C09131=1138.833,163.232,-60.014,-178.582,7.169,148.928
C09132=1138.829,163.481,-60.036,-178.579,7.171,148.927
C09133=1138.824,163.730,-60.058,-178.576,7.174,148.927
C09134=1138.820,163.979,-60.080,-178.574,7.176,148.927
C09135=1138.815,164.228,-60.102,-178.571,7.177,148.926
C09136=1138.810,164.478,-60.124,-178.568,7.180,148.926
C09137=1138.805,164.726,-60.146,-178.565,7.182,148.926
C09138=1138.801,164.975,-60.169,-178.562,7.185,148.925
C09139=1138.796,165.224,-60.191,-178.560,7.186,148.925
C09140=1138.792,165.473,-60.213,-178.557,7.188,148.925
C09141=1138.787,165.722,-60.234,-178.554,7.191,148.924
C09142=1138.782,165.971,-60.257,-178.551,7.193,148.924
C09143=1138.777,166.220,-60.279,-178.548,7.195,148.924
C09144=1138.773,166.469,-60.301,-178.545,7.197,148.923
C09145=1138.769,166.717,-60.323,-178.543,7.200,148.923
C09146=1138.764,166.967,-60.346,-178.540,7.201,148.923
C09147=1138.759,167.216,-60.367,-178.537,7.203,148.923
C09148=1138.754,167.465,-60.390,-178.534,7.206,148.922
C09149=1138.750,167.714,-60.412,-178.532,7.208,148.922
C09150=1138.745,167.963,-60.435,-178.528,7.210,148.922
C09151=1138.741,168.212,-60.457,-178.526,7.212,148.921
C09152=1138.736,168.461,-60.478,-178.523,7.215,148.921
C09153=1138.731,168.710,-60.501,-178.520,7.217,148.921
C09154=1138.726,168.958,-60.523,-178.518,7.219,148.921
C09155=1138.722,169.208,-60.545,-178.515,7.221,148.920
C09156=1138.718,169.457,-60.567,-178.512,7.223,148.920
C09157=1138.712,169.705,-60.590,-178.509,7.226,148.920
C09158=1138.708,169.955,-60.612,-178.506,7.228,148.919
C09159=1138.703,170.203,-60.634,-178.503,7.230,148.919
C09160=1138.698,170.452,-60.657,-178.500,7.232,148.919
C09161=1138.694,170.702,-60.680,-178.497,7.235,148.919
C09162=1138.689,170.951,-60.702,-178.495,7.236,148.918
C09163=1138.685,171.199,-60.725,-178.492,7.239,148.918
C09164=1138.680,171.448,-60.746,-178.489,7.241,148.918
C09165=1138.675,171.697,-60.770,-178.487,7.243,148.917
C09166=1138.671,171.946,-60.792,-178.484,7.246,148.917
C09167=1138.665,172.195,-60.814,-178.481,7.247,148.917
C09168=1138.661,172.444,-60.837,-178.478,7.250,148.916
C09169=1138.657,172.693,-60.859,-178.475,7.252,148.916
C09170=1138.652,172.942,-60.882,-178.472,7.254,148.916
C09171=1138.647,173.191,-60.904,-178.469,7.256,148.916
C09172=1138.643,173.440,-60.927,-178.467,7.259,148.915
C09173=1138.638,173.689,-60.949,-178.464,7.261,148.915
C09174=1138.633,173.938,-60.972,-178.461,7.263,148.915
C09175=1138.629,174.187,-60.994,-178.458,7.265,148.915
C09176=1138.624,174.435,-61.017,-178.455,7.268,148.914
C09177=1138.620,174.684,-61.040,-178.452,7.270,148.914
C09178=1138.615,174.934,-61.063,-178.450,7.273,148.914
C09179=1138.610,175.182,-61.085,-178.447,7.274,148.913
C09180=1138.605,175.431,-61.108,-178.444,7.277,148.913
C09181=1138.601,175.680,-61.130,-178.441,7.279,148.913
C09182=1138.596,175.929,-61.154,-178.438,7.281,148.912
C09183=1138.591,176.178,-61.176,-178.436,7.284,148.912
C09184=1138.587,176.427,-61.199,-178.433,7.286,148.912
C09185=1138.583,176.676,-61.222,-178.430,7.288,148.912
C09186=1138.578,176.925,-61.244,-178.427,7.291,148.912
C09187=1138.573,177.173,-61.267,-178.424,7.292,148.911
C09188=1138.569,177.422,-61.290,-178.422,7.295,148.911
C09189=1138.563,177.672,-61.313,-178.419,7.297,148.911
C09190=1138.560,177.921,-61.335,-178.416,7.300,148.910
C09191=1138.554,178.169,-61.358,-178.413,7.302,148.910
C09192=1138.550,178.418,-61.381,-178.410,7.304,148.910
C09193=1138.545,178.667,-61.404,-178.408,7.306,148.910
C09194=1138.541,178.916,-61.427,-178.404,7.309,148.909
C09195=1138.537,179.165,-61.450,-178.402,7.310,148.909
C09196=1138.531,179.413,-61.473,-178.399,7.313,148.909
C09197=1138.527,179.662,-61.496,-178.396,7.315,148.908
C09198=1138.522,179.912,-61.518,-178.393,7.318,148.908
C09199=1138.518,180.161,-61.542,-178.390,7.321,148.908
C09200=1138.514,180.410,-61.564,-178.388,7.323,148.908
C09201=1138.509,180.659,-61.588,-178.385,7.325,148.907
C09202=1138.504,180.907,-61.611,-178.382,7.327,148.907
C09203=1138.499,181.156,-61.634,-178.379,7.330,148.907
C09204=1138.495,181.405,-61.657,-178.376,7.331,148.907
C09205=1138.490,181.654,-61.680,-178.374,7.334,148.907
C09206=1138.485,181.903,-61.703,-178.371,7.336,148.906
C09207=1138.481,182.152,-61.726,-178.368,7.339,148.906
C09208=1138.477,182.401,-61.749,-178.365,7.341,148.906
C09209=1138.471,182.649,-61.772,-178.362,7.343,148.905
C09210=1138.467,182.898,-61.795,-178.359,7.346,148.905
C09211=1138.462,183.167,-61.821,-178.357,7.348,148.905
C09212=1138.458,183.438,-61.846,-178.354,7.351,148.905
C09213=1138.452,183.708,-61.871,-178.350,7.353,148.904
C09214=1138.447,183.977,-61.896,-178.347,7.356,148.904
C09215=1138.442,184.226,-61.919,-178.344,7.359,148.904
C09216=1138.438,184.475,-61.942,-178.342,7.360,148.904
C09217=1138.434,184.724,-61.966,-178.339,7.363,148.903
C09218=1138.429,184.972,-61.990,-178.336,7.365,148.903
C09219=1138.424,185.221,-62.013,-178.333,7.368,148.903
C09220=1138.419,185.470,-62.036,-178.331,7.370,148.903
C09221=1138.415,185.719,-62.059,-178.327,7.372,148.902
C09222=1138.411,185.968,-62.082,-178.325,7.375,148.902
C09223=1138.406,186.217,-62.105,-178.322,7.377,148.902
C09224=1138.401,186.466,-62.129,-178.319,7.380,148.902
C09225=1138.396,186.715,-62.152,-178.316,7.381,148.901
C09226=1138.392,186.963,-62.176,-178.314,7.384,148.901
C09227=1138.387,187.212,-62.200,-178.310,7.387,148.901
C09228=1138.383,187.461,-62.223,-178.308,7.389,148.901
C09229=1138.378,187.710,-62.246,-178.305,7.392,148.900
C09230=1138.374,187.959,-62.270,-178.302,7.394,148.900
C09231=1138.369,188.208,-62.294,-178.299,7.396,148.900
C09232=1138.364,188.457,-62.317,-178.296,7.399,148.900
C09233=1138.360,188.706,-62.340,-178.294,7.401,148.899
C09234=1138.355,188.954,-62.365,-178.291,7.404,148.899
C09235=1138.350,189.203,-62.388,-178.288,7.405,148.899
C09236=1138.346,189.452,-62.411,-178.285,7.408,148.899
C09237=1138.341,189.701,-62.435,-178.282,7.411,148.898
C09238=1138.337,189.950,-62.459,-178.280,7.413,148.898
C09239=1138.332,190.199,-62.482,-178.277,7.415,148.898
C09240=1138.328,190.447,-62.506,-178.274,7.418,148.898
C09241=1138.323,190.696,-62.529,-178.271,7.420,148.898
C09242=1138.318,190.945,-62.553,-178.268,7.423,148.897
C09243=1138.314,191.194,-62.577,-178.266,7.425,148.897
C09244=1138.309,191.443,-62.600,-178.263,7.428,148.897
C09245=1138.305,191.691,-62.624,-178.259,7.430,148.897
C09246=1138.300,191.940,-62.648,-178.257,7.432,148.896
C09247=1138.295,192.189,-62.671,-178.254,7.435,148.896
C09248=1138.291,192.437,-62.695,-178.252,7.437,148.896
C09249=1138.287,192.687,-62.719,-178.248,7.439,148.896
C09250=1138.282,192.936,-62.743,-178.246,7.442,148.896
C09251=1138.278,193.185,-62.766,-178.243,7.444,148.895
C09252=1138.273,193.433,-62.790,-178.240,7.447,148.895
C09253=1138.268,193.682,-62.814,-178.237,7.450,148.895
C09254=1138.263,193.931,-62.838,-178.235,7.452,148.895
C09255=1138.259,194.180,-62.862,-178.232,7.454,148.894
C09256=1138.254,194.428,-62.886,-178.228,7.457,148.894
C09257=1138.250,194.677,-62.910,-178.226,7.459,148.894
C09258=1138.246,194.926,-62.934,-178.223,7.462,148.894
C09259=1138.241,195.175,-62.958,-178.220,7.464,148.894
C09260=1138.236,195.424,-62.982,-178.218,7.467,148.893
C09261=1138.232,195.673,-63.006,-178.215,7.469,148.893
C09262=1138.227,195.921,-63.030,-178.212,7.472,148.893
C09263=1138.223,196.170,-63.053,-178.209,7.474,148.893
C09264=1138.217,196.419,-63.078,-178.206,7.477,148.892
C09265=1138.214,196.668,-63.102,-178.203,7.479,148.892
C09266=1138.209,196.917,-63.126,-178.201,7.481,148.892
C09267=1138.205,197.165,-63.150,-178.198,7.484,148.892
C09268=1138.199,197.414,-63.174,-178.195,7.487,148.892
C09269=1138.195,197.662,-63.198,-178.193,7.489,148.891
C09270=1138.191,197.912,-63.222,-178.189,7.491,148.891
C09271=1138.186,198.161,-63.246,-178.186,7.494,148.891
C09272=1138.181,198.409,-63.271,-178.184,7.496,148.891
C09273=1138.177,198.658,-63.295,-178.181,7.499,148.891
C09274=1138.172,198.907,-63.318,-178.178,7.502,148.890
C09275=1138.168,199.156,-63.343,-178.175,7.504,148.890
C09276=1138.163,199.405,-63.367,-178.173,7.506,148.890
C09277=1138.159,199.653,-63.392,-178.169,7.509,148.890
C09278=1138.155,199.901,-63.416,-178.167,7.511,148.889
C09279=1138.150,200.151,-63.441,-178.164,7.514,148.889
C09280=1138.145,200.400,-63.464,-178.161,7.516,148.889
C09281=1138.140,200.649,-63.489,-178.159,7.519,148.889
C09282=1138.136,200.897,-63.513,-178.156,7.521,148.889
C09283=1138.132,201.146,-63.537,-178.153,7.524,148.888
C09284=1138.127,201.395,-63.562,-178.150,7.527,148.888
C09285=1138.122,201.643,-63.586,-178.147,7.529,148.888
C09286=1138.118,201.892,-63.610,-178.144,7.532,148.888
C09287=1138.114,202.141,-63.635,-178.142,7.534,148.888
C09288=1138.109,202.390,-63.659,-178.139,7.536,148.887
C09289=1138.104,202.638,-63.684,-178.136,7.539,148.887
C09290=1138.100,202.887,-63.708,-178.133,7.542,148.887
C09291=1138.095,203.136,-63.733,-178.130,7.545,148.887
C09292=1138.091,203.384,-63.757,-178.128,7.547,148.887
C09293=1138.087,203.634,-63.781,-178.125,7.550,148.887
C09294=1138.082,203.882,-63.806,-178.122,7.552,148.886
C09295=1138.077,204.131,-63.830,-178.119,7.555,148.886
C09296=1138.073,204.380,-63.855,-178.116,7.557,148.886
C09297=1138.068,204.629,-63.879,-178.113,7.560,148.886
C09298=1138.063,204.877,-63.904,-178.111,7.563,148.886
C09299=1138.060,205.126,-63.929,-178.108,7.564,148.885
C09300=1138.055,205.375,-63.954,-178.105,7.567,148.885
C09301=1138.050,205.623,-63.978,-178.102,7.570,148.885
C09302=1138.046,205.872,-64.003,-178.099,7.573,148.885
C09303=1138.041,206.121,-64.028,-178.097,7.575,148.885
C09304=1138.036,206.369,-64.052,-178.094,7.578,148.885
C09305=1138.032,206.619,-64.077,-178.091,7.580,148.884
C09306=1138.028,206.867,-64.101,-178.088,7.583,148.884
C09307=1138.023,207.116,-64.126,-178.086,7.585,148.884
C09308=1138.018,207.365,-64.151,-178.083,7.588,148.884
C09309=1138.014,207.613,-64.175,-178.080,7.591,148.884
C09310=1138.009,207.862,-64.201,-178.077,7.593,148.883
C09311=1138.005,208.110,-64.225,-178.074,7.596,148.883
C09312=1138.000,208.360,-64.250,-178.071,7.598,148.883
C09313=1137.996,208.608,-64.275,-178.068,7.601,148.883
C09314=1137.991,208.856,-64.300,-178.066,7.604,148.883
C09315=1137.986,209.128,-64.327,-178.062,7.606,148.882
C09316=1137.981,209.398,-64.354,-178.059,7.609,148.882
C09317=1137.976,209.669,-64.381,-178.056,7.612,148.882
C09318=1137.972,209.940,-64.408,-178.053,7.615,148.882
C09319=1137.967,210.188,-64.433,-178.051,7.618,148.882
C09320=1137.962,210.437,-64.459,-178.047,7.620,148.882
C09321=1137.958,210.685,-64.483,-178.045,7.622,148.881
C09322=1137.954,210.934,-64.508,-178.042,7.625,148.881
C09323=1137.949,211.183,-64.533,-178.039,7.628,148.881
C09324=1137.945,211.432,-64.557,-178.036,7.631,148.881
C09325=1137.940,211.680,-64.583,-178.033,7.634,148.881
C09326=1137.935,211.930,-64.608,-178.031,7.636,148.881
C09327=1137.931,212.178,-64.633,-178.028,7.639,148.881
C09328=1137.926,212.427,-64.658,-178.025,7.641,148.880
C09329=1137.922,212.675,-64.683,-178.022,7.644,148.880
C09330=1137.917,212.924,-64.708,-178.019,7.647,148.880
C09331=1137.913,213.172,-64.733,-178.017,7.649,148.880
C09332=1137.908,213.421,-64.759,-178.014,7.652,148.880
C09333=1137.904,213.670,-64.783,-178.011,7.655,148.879
C09334=1137.900,213.919,-64.809,-178.008,7.657,148.879
C09335=1137.895,214.168,-64.834,-178.006,7.660,148.879
C09336=1137.890,214.416,-64.859,-178.003,7.662,148.879
C09337=1137.886,214.665,-64.885,-178.000,7.665,148.879
C09338=1137.881,214.914,-64.910,-177.997,7.668,148.879
C09339=1137.877,215.162,-64.936,-177.994,7.671,148.879
C09340=1137.872,215.411,-64.960,-177.991,7.673,148.878
C09341=1137.868,215.660,-64.985,-177.988,7.676,148.878
C09342=1137.864,215.908,-65.011,-177.986,7.678,148.878
C09343=1137.859,216.156,-65.037,-177.983,7.681,148.878
C09344=1137.855,216.406,-65.062,-177.981,7.684,148.878
C09345=1137.850,216.654,-65.087,-177.977,7.687,148.878
C09346=1137.846,216.903,-65.113,-177.974,7.690,148.878
C09347=1137.841,217.152,-65.138,-177.972,7.692,148.877
C09348=1137.836,217.400,-65.163,-177.969,7.695,148.877
C09349=1137.832,217.649,-65.189,-177.966,7.697,148.877
C09350=1137.827,217.897,-65.214,-177.963,7.700,148.877
C09351=1137.823,218.146,-65.240,-177.961,7.703,148.877
C09352=1137.818,218.396,-65.265,-177.958,7.706,148.877
C09353=1137.814,218.643,-65.290,-177.955,7.709,148.877
C09354=1137.810,218.892,-65.316,-177.952,7.711,148.876
C09355=1137.806,219.141,-65.341,-177.949,7.713,148.876
C09356=1137.801,219.389,-65.367,-177.947,7.716,148.876
C09357=1137.797,219.638,-65.393,-177.944,7.719,148.876
C09358=1137.792,219.887,-65.419,-177.941,7.722,148.876
C09359=1137.787,220.135,-65.444,-177.938,7.725,148.876
C09360=1137.783,220.384,-65.469,-177.935,7.728,148.875
C09361=1137.778,220.633,-65.495,-177.933,7.730,148.875
C09362=1137.774,220.882,-65.521,-177.930,7.733,148.875
C09363=1137.769,221.130,-65.546,-177.927,7.735,148.875
C09364=1137.765,221.379,-65.572,-177.924,7.738,148.875
C09365=1137.761,221.628,-65.598,-177.921,7.741,148.875
C09366=1137.756,221.876,-65.623,-177.918,7.744,148.875
C09367=1137.752,222.125,-65.649,-177.915,7.747,148.875
C09368=1137.748,222.373,-65.675,-177.913,7.749,148.874
C09369=1137.743,222.622,-65.700,-177.910,7.752,148.874
C09370=1137.738,222.871,-65.726,-177.908,7.755,148.874
C09371=1137.734,223.119,-65.753,-177.905,7.758,148.874
C09372=1137.730,223.368,-65.779,-177.901,7.760,148.874
C09373=1137.725,223.616,-65.804,-177.899,7.763,148.874
C09374=1137.721,223.865,-65.830,-177.896,7.766,148.874
C09375=1137.716,224.113,-65.855,-177.893,7.769,148.874
C09376=1137.711,224.363,-65.882,-177.891,7.771,148.873
C09377=1137.707,224.611,-65.908,-177.888,7.774,148.873
C09378=1137.702,224.859,-65.933,-177.885,7.777,148.873
C09379=1137.698,225.108,-65.959,-177.882,7.780,148.873
C09380=1137.694,225.356,-65.985,-177.879,7.782,148.873
C09381=1137.689,225.606,-66.011,-177.876,7.785,148.873
C09382=1137.685,225.854,-66.037,-177.874,7.788,148.873
C09383=1137.680,226.102,-66.063,-177.871,7.791,148.873
C09384=1137.676,226.351,-66.089,-177.868,7.794,148.872
C09385=1137.671,226.600,-66.115,-177.865,7.797,148.872
C09386=1137.667,226.849,-66.141,-177.863,7.799,148.872
C09387=1137.663,227.097,-66.167,-177.860,7.802,148.872
C09388=1137.658,227.345,-66.194,-177.857,7.804,148.872
C09389=1137.653,227.594,-66.219,-177.854,7.807,148.872
C09390=1137.649,227.843,-66.245,-177.851,7.810,148.872
C09391=1137.645,228.091,-66.272,-177.848,7.813,148.872
C09392=1137.640,228.340,-66.298,-177.846,7.816,148.872
C09393=1137.636,228.589,-66.324,-177.843,7.819,148.871
C09394=1137.632,228.837,-66.350,-177.840,7.822,148.871
C09395=1137.627,229.086,-66.377,-177.837,7.825,148.871
C09396=1137.623,229.334,-66.403,-177.834,7.828,148.871
C09397=1137.618,229.583,-66.429,-177.832,7.830,148.871
C09398=1137.613,229.832,-66.455,-177.829,7.833,148.871
C09399=1137.609,230.080,-66.481,-177.826,7.835,148.871
C09400=1137.605,230.329,-66.508,-177.823,7.838,148.871
C09401=1137.601,230.577,-66.534,-177.821,7.841,148.870
C09402=1137.596,230.826,-66.560,-177.818,7.844,148.870
C09403=1137.592,231.074,-66.587,-177.815,7.847,148.870
C09404=1137.587,231.323,-66.613,-177.812,7.850,148.870
C09405=1137.583,231.572,-66.640,-177.809,7.853,148.870
C09406=1137.579,231.820,-66.665,-177.806,7.855,148.870
C09407=1137.573,232.068,-66.692,-177.804,7.858,148.870
C09408=1137.569,232.316,-66.719,-177.801,7.861,148.870
C09409=1137.564,232.566,-66.745,-177.798,7.864,148.870
C09410=1137.561,232.814,-66.771,-177.795,7.867,148.870
C09411=1137.556,233.063,-66.798,-177.792,7.870,148.870
C09412=1137.552,233.311,-66.824,-177.790,7.873,148.870
C09413=1137.547,233.560,-66.851,-177.787,7.876,148.869
C09414=1137.543,233.808,-66.877,-177.784,7.879,148.869
C09415=1137.538,234.057,-66.904,-177.782,7.881,148.869
C09416=1137.534,234.305,-66.930,-177.779,7.883,148.869
C09417=1137.529,234.554,-66.957,-177.776,7.886,148.869
C09418=1137.525,234.802,-66.983,-177.773,7.889,148.869
C09419=1137.521,235.075,-67.013,-177.770,7.893,148.869
C09420=1137.515,235.347,-67.042,-177.767,7.896,148.869
C09421=1137.510,235.618,-67.071,-177.764,7.899,148.869
C09422=1137.506,235.890,-67.100,-177.761,7.902,148.869
C09423=1137.502,236.139,-67.127,-177.758,7.905,148.868
C09424=1137.497,236.388,-67.154,-177.755,7.908,148.868
C09425=1137.493,236.636,-67.180,-177.752,7.911,148.868
C09426=1137.488,236.885,-67.207,-177.749,7.914,148.868
C09427=1137.484,237.133,-67.234,-177.747,7.917,148.868
C09428=1137.480,237.381,-67.261,-177.744,7.920,148.868
C09429=1137.475,237.630,-67.288,-177.741,7.923,148.868
C09430=1137.470,237.879,-67.314,-177.738,7.926,148.868
C09431=1137.466,238.127,-67.340,-177.736,7.928,148.868
C09432=1137.461,238.376,-67.368,-177.733,7.931,148.868
C09433=1137.457,238.624,-67.395,-177.730,7.934,148.868
C09434=1137.453,238.872,-67.421,-177.728,7.937,148.867
C09435=1137.448,239.121,-67.448,-177.725,7.940,148.867
C09436=1137.444,239.369,-67.475,-177.722,7.942,148.867
C09437=1137.440,239.618,-67.502,-177.719,7.945,148.867
C09438=1137.436,239.867,-67.529,-177.716,7.948,148.867
C09439=1137.431,240.115,-67.556,-177.714,7.951,148.867
C09440=1137.426,240.364,-67.583,-177.711,7.954,148.867
C09441=1137.422,240.612,-67.610,-177.708,7.957,148.867
C09442=1137.418,240.860,-67.637,-177.705,7.960,148.867
C09443=1137.413,241.109,-67.664,-177.702,7.963,148.867
C09444=1137.409,241.358,-67.691,-177.700,7.966,148.867
C09445=1137.404,241.607,-67.718,-177.697,7.969,148.867
C09446=1137.400,241.855,-67.745,-177.694,7.972,148.867
C09447=1137.396,242.103,-67.772,-177.691,7.974,148.866
C09448=1137.391,242.352,-67.799,-177.688,7.977,148.866
C09449=1137.387,242.600,-67.827,-177.686,7.980,148.866
C09450=1137.383,242.849,-67.854,-177.682,7.984,148.866
C09451=1137.378,243.097,-67.881,-177.679,7.987,148.866
C09452=1137.374,243.346,-67.908,-177.677,7.990,148.866
C09453=1137.370,243.594,-67.935,-177.674,7.993,148.866
C09454=1137.365,243.843,-67.962,-177.671,7.996,148.866
C09455=1137.361,244.091,-67.990,-177.668,7.999,148.866
C09456=1137.356,244.340,-68.017,-177.666,8.002,148.866
C09457=1137.352,244.588,-68.044,-177.663,8.005,148.866
C09458=1137.347,244.837,-68.071,-177.660,8.008,148.866
C09459=1137.343,245.084,-68.099,-177.657,8.011,148.866
C09460=1137.339,245.334,-68.126,-177.655,8.013,148.866
C09461=1137.334,245.582,-68.153,-177.652,8.016,148.866
C09462=1137.329,245.831,-68.180,-177.649,8.019,148.866
C09463=1137.325,246.079,-68.208,-177.646,8.022,148.865
C09464=1137.322,246.327,-68.235,-177.643,8.025,148.865
C09465=1137.317,246.576,-68.262,-177.641,8.028,148.865
C09466=1137.313,246.824,-68.290,-177.638,8.031,148.865
C09467=1137.308,247.072,-68.317,-177.635,8.034,148.865
C09468=1137.304,247.321,-68.345,-177.632,8.037,148.865
C09469=1137.300,247.569,-68.372,-177.629,8.040,148.865
C09470=1137.294,247.818,-68.400,-177.627,8.043,148.865
C09471=1137.291,248.067,-68.428,-177.624,8.046,148.865
C09472=1137.286,248.315,-68.455,-177.621,8.049,148.865
C09473=1137.282,248.563,-68.483,-177.619,8.052,148.865
C09474=1137.277,248.812,-68.510,-177.616,8.055,148.865
C09475=1137.273,249.060,-68.538,-177.613,8.057,148.865
C09476=1137.268,249.309,-68.565,-177.610,8.061,148.865
C09477=1137.264,249.557,-68.593,-177.607,8.064,148.865
C09478=1137.260,249.806,-68.620,-177.604,8.067,148.865
C09479=1137.256,250.054,-68.648,-177.601,8.070,148.864
C09480=1137.252,250.303,-68.675,-177.599,8.073,148.865
C09481=1137.247,250.551,-68.703,-177.596,8.076,148.865
C09482=1137.243,250.799,-68.730,-177.593,8.079,148.864
C09483=1137.238,251.048,-68.759,-177.590,8.082,148.864
C09484=1137.234,251.296,-68.787,-177.588,8.085,148.864
C09485=1137.229,251.544,-68.814,-177.585,8.088,148.864
C09486=1137.225,251.793,-68.842,-177.582,8.091,148.864
C09487=1137.221,252.041,-68.870,-177.579,8.094,148.864
C09488=1137.216,252.289,-68.897,-177.577,8.097,148.864
C09489=1137.212,252.538,-68.926,-177.574,8.100,148.864
C09490=1137.208,252.786,-68.953,-177.571,8.103,148.864
C09491=1137.203,253.035,-68.981,-177.568,8.106,148.864
C09492=1137.199,253.283,-69.009,-177.565,8.109,148.864
C09493=1137.195,253.532,-69.037,-177.562,8.112,148.864
C09494=1137.190,253.781,-69.064,-177.560,8.115,148.864
C09495=1137.186,254.028,-69.092,-177.557,8.118,148.864
C09496=1137.182,254.277,-69.120,-177.554,8.121,148.864
C09497=1137.178,254.525,-69.148,-177.552,8.124,148.864
C09498=1137.173,254.774,-69.177,-177.549,8.127,148.864
C09499=1137.168,255.022,-69.204,-177.546,8.130,148.864
C09500=1137.165,255.271,-69.232,-177.543,8.133,148.864
C09501=1137.160,255.519,-69.260,-177.540,8.137,148.864
C09502=1137.156,255.768,-69.288,-177.538,8.140,148.864
C09503=1137.151,256.016,-69.316,-177.535,8.143,148.864
C09504=1137.146,256.264,-69.345,-177.532,8.146,148.864
C09505=1137.143,256.512,-69.373,-177.529,8.149,148.864
C09506=1137.138,256.760,-69.401,-177.526,8.152,148.864
C09507=1137.133,257.010,-69.429,-177.524,8.155,148.864
C09508=1137.129,257.258,-69.456,-177.521,8.158,148.864
C09509=1137.125,257.506,-69.484,-177.518,8.161,148.864
C09510=1137.120,257.754,-69.513,-177.515,8.164,148.863
C09511=1137.117,258.003,-69.541,-177.512,8.167,148.863
C09512=1137.112,258.252,-69.570,-177.510,8.171,148.864
C09513=1137.108,258.500,-69.597,-177.507,8.174,148.863
C09514=1137.104,258.748,-69.626,-177.504,8.176,148.863
C09515=1137.099,258.996,-69.654,-177.501,8.179,148.863
C09516=1137.095,259.245,-69.682,-177.499,8.182,148.863
C09517=1137.090,259.493,-69.711,-177.496,8.186,148.863
C09518=1137.087,259.741,-69.739,-177.493,8.189,148.863
C09519=1137.081,259.989,-69.768,-177.490,8.192,148.863
C09520=1137.078,260.238,-69.796,-177.487,8.195,148.863
C09521=1137.073,260.486,-69.824,-177.485,8.198,148.863
C09522=1137.069,260.735,-69.852,-177.482,8.201,148.863
C09523=1137.064,261.008,-69.883,-177.479,8.205,148.863
C09524=1137.060,261.282,-69.915,-177.476,8.208,148.863
C09525=1137.054,261.555,-69.947,-177.473,8.212,148.863
C09526=1137.050,261.829,-69.978,-177.470,8.215,148.863
C09527=1137.045,262.078,-70.006,-177.467,8.218,148.863
C09528=1137.042,262.326,-70.035,-177.464,8.222,148.863
C09529=1137.037,262.574,-70.063,-177.461,8.224,148.863
C09530=1137.033,262.822,-70.092,-177.459,8.227,148.863
C09531=1137.028,263.071,-70.120,-177.456,8.231,148.863
C09532=1137.024,263.318,-70.149,-177.453,8.234,148.863
C09533=1137.020,263.567,-70.177,-177.451,8.236,148.863
C09534=1137.015,263.816,-70.206,-177.447,8.240,148.863
C09535=1137.011,264.063,-70.235,-177.445,8.243,148.863
C09536=1137.007,264.312,-70.263,-177.442,8.246,148.863
C09537=1137.002,264.561,-70.292,-177.439,8.249,148.863
C09538=1136.998,264.809,-70.321,-177.436,8.252,148.863
C09539=1136.994,265.057,-70.349,-177.434,8.255,148.863
C09540=1136.990,265.306,-70.378,-177.431,8.258,148.863
C09541=1136.985,265.554,-70.407,-177.428,8.262,148.863
C09542=1136.981,265.802,-70.435,-177.425,8.265,148.863
C09543=1136.977,266.051,-70.465,-177.423,8.268,148.863
C09544=1136.972,266.299,-70.493,-177.420,8.271,148.863
C09545=1136.968,266.547,-70.522,-177.417,8.274,148.863
C09546=1136.964,266.796,-70.551,-177.414,8.278,148.863
C09547=1136.959,267.044,-70.579,-177.411,8.281,148.863
C09548=1136.955,267.292,-70.608,-177.409,8.284,148.863
C09549=1136.951,267.541,-70.637,-177.406,8.287,148.863
C09550=1136.946,267.789,-70.666,-177.404,8.290,148.863
C09551=1136.942,268.036,-70.695,-177.401,8.293,148.863
C09552=1136.938,268.285,-70.723,-177.397,8.297,148.863
C09553=1136.934,268.533,-70.753,-177.395,8.300,148.863
C09554=1136.929,268.782,-70.782,-177.392,8.303,148.863
C09555=1136.925,269.030,-70.810,-177.389,8.306,148.863
C09556=1136.921,269.278,-70.840,-177.387,8.309,148.863
C09557=1136.917,269.527,-70.868,-177.384,8.313,148.863
C09558=1136.912,269.775,-70.898,-177.381,8.316,148.863
C09559=1136.907,270.023,-70.926,-177.379,8.319,148.863
C09560=1136.903,270.271,-70.956,-177.376,8.322,148.863
C09561=1136.900,270.519,-70.984,-177.373,8.325,148.863
C09562=1136.895,270.768,-71.014,-177.370,8.329,148.864
C09563=1136.891,271.017,-71.043,-177.367,8.332,148.863
C09564=1136.886,271.264,-71.072,-177.364,8.335,148.863
C09565=1136.882,271.512,-71.101,-177.362,8.338,148.864
C09566=1136.877,271.761,-71.130,-177.359,8.341,148.864
C09567=1136.873,272.010,-71.159,-177.356,8.345,148.863
C09568=1136.869,272.258,-71.189,-177.354,8.348,148.864
C09569=1136.866,272.506,-71.218,-177.351,8.351,148.864
C09570=1136.861,272.753,-71.247,-177.348,8.354,148.864
C09571=1136.857,273.002,-71.276,-177.346,8.357,148.864
C09572=1136.852,273.251,-71.305,-177.342,8.361,148.864
C09573=1136.848,273.499,-71.334,-177.339,8.364,148.864
C09574=1136.844,273.747,-71.364,-177.337,8.367,148.864
C09575=1136.840,273.995,-71.393,-177.334,8.370,148.864
C09576=1136.836,274.244,-71.423,-177.331,8.374,148.864
C09577=1136.831,274.492,-71.452,-177.329,8.377,148.864
C09578=1136.827,274.739,-71.481,-177.326,8.380,148.864
C09579=1136.822,274.988,-71.511,-177.323,8.383,148.864
C09580=1136.818,275.236,-71.540,-177.320,8.387,148.864
C09581=1136.814,275.484,-71.570,-177.317,8.390,148.864
C09582=1136.810,275.732,-71.599,-177.315,8.393,148.864
C09583=1136.806,275.981,-71.629,-177.312,8.396,148.864
C09584=1136.801,276.229,-71.658,-177.310,8.399,148.864
C09585=1136.797,276.477,-71.688,-177.306,8.403,148.864
C09586=1136.793,276.726,-71.717,-177.304,8.406,148.864
C09587=1136.789,276.974,-71.746,-177.301,8.409,148.864
C09588=1136.784,277.222,-71.776,-177.299,8.412,148.864
C09589=1136.780,277.471,-71.806,-177.296,8.416,148.864
C09590=1136.776,277.719,-71.835,-177.293,8.419,148.864
C09591=1136.771,277.967,-71.865,-177.290,8.422,148.864
C09592=1136.767,278.215,-71.894,-177.288,8.425,148.864
C09593=1136.763,278.464,-71.924,-177.284,8.429,148.864
C09594=1136.759,278.711,-71.954,-177.282,8.432,148.865
C09595=1136.755,278.960,-71.983,-177.279,8.435,148.865
C09596=1136.751,279.208,-72.013,-177.277,8.438,148.865
C09597=1136.746,279.457,-72.043,-177.273,8.442,148.865
C09598=1136.742,279.705,-72.072,-177.271,8.445,148.865
C09599=1136.738,279.952,-72.102,-177.268,8.448,148.865
C09600=1136.734,280.201,-72.132,-177.265,8.452,148.865
C09601=1136.730,280.449,-72.161,-177.263,8.455,148.865
C09602=1136.725,280.698,-72.191,-177.260,8.458,148.865
C09603=1136.721,280.945,-72.222,-177.257,8.461,148.865
C09604=1136.717,281.193,-72.251,-177.254,8.465,148.865
C09605=1136.712,281.442,-72.281,-177.252,8.468,148.865
C09606=1136.708,281.690,-72.311,-177.249,8.471,148.865
C09607=1136.704,281.938,-72.341,-177.247,8.475,148.865
C09608=1136.699,282.186,-72.370,-177.243,8.478,148.865
C09609=1136.695,282.434,-72.400,-177.241,8.481,148.865
C09610=1136.691,282.682,-72.430,-177.238,8.484,148.865
C09611=1136.686,282.931,-72.460,-177.235,8.488,148.866
C09612=1136.683,283.178,-72.490,-177.232,8.491,148.866
C09613=1136.678,283.427,-72.520,-177.230,8.495,148.866
C09614=1136.674,283.675,-72.550,-177.227,8.498,148.866
C09615=1136.670,283.923,-72.580,-177.224,8.502,148.866
C09616=1136.666,284.172,-72.611,-177.221,8.505,148.866
C09617=1136.661,284.420,-72.640,-177.219,8.508,148.866
C09618=1136.657,284.667,-72.670,-177.216,8.512,148.866
C09619=1136.653,284.916,-72.700,-177.213,8.515,148.866
C09620=1136.649,285.164,-72.731,-177.211,8.518,148.866
C09621=1136.644,285.412,-72.761,-177.208,8.522,148.866
C09622=1136.640,285.660,-72.791,-177.205,8.525,148.866
C09623=1136.636,285.908,-72.820,-177.203,8.528,148.866
C09624=1136.632,286.157,-72.851,-177.200,8.531,148.866
C09625=1136.628,286.404,-72.882,-177.197,8.535,148.867
C09626=1136.623,286.653,-72.912,-177.194,8.538,148.866
C09627=1136.619,286.928,-72.945,-177.191,8.542,148.867
C09628=1136.613,287.204,-72.979,-177.188,8.546,148.867
C09629=1136.609,287.480,-73.012,-177.185,8.549,148.867
C09630=1136.604,287.755,-73.047,-177.182,8.553,148.867
C09631=1136.600,288.004,-73.076,-177.179,8.557,148.867
C09632=1136.596,288.252,-73.107,-177.176,8.560,148.867
C09633=1136.592,288.499,-73.137,-177.174,8.563,148.867
C09634=1136.588,288.748,-73.168,-177.171,8.567,148.867
C09635=1136.583,288.996,-73.197,-177.168,8.570,148.867
C09636=1136.579,289.244,-73.228,-177.166,8.573,148.867
C09637=1136.575,289.492,-73.258,-177.162,8.577,148.867
C09638=1136.570,289.740,-73.289,-177.160,8.580,148.868
C09639=1136.567,289.988,-73.320,-177.157,8.583,148.868
C09640=1136.562,290.237,-73.350,-177.154,8.587,148.868
C09641=1136.558,290.484,-73.380,-177.152,8.590,148.868
C09642=1136.554,290.732,-73.411,-177.149,8.593,148.868
C09643=1136.550,290.981,-73.442,-177.146,8.597,148.868
C09644=1136.546,291.229,-73.472,-177.144,8.600,148.868
C09645=1136.541,291.477,-73.503,-177.141,8.604,148.868
C09646=1136.538,291.725,-73.533,-177.138,8.608,148.868
C09647=1136.533,291.973,-73.564,-177.135,8.611,148.868
C09648=1136.529,292.221,-73.595,-177.133,8.614,148.869
C09649=1136.525,292.469,-73.624,-177.130,8.618,148.869
C09650=1136.521,292.718,-73.655,-177.127,8.621,148.869
C09651=1136.516,292.966,-73.686,-177.125,8.624,148.869
C09652=1136.512,293.213,-73.716,-177.122,8.628,148.869
C09653=1136.508,293.462,-73.747,-177.119,8.631,148.869
C09654=1136.503,293.710,-73.778,-177.117,8.634,148.869
C09655=1136.500,293.957,-73.809,-177.114,8.638,148.869
C09656=1136.496,294.206,-73.840,-177.111,8.641,148.869
C09657=1136.491,294.454,-73.871,-177.108,8.645,148.870
C09658=1136.487,294.701,-73.901,-177.106,8.648,148.870
C09659=1136.483,294.950,-73.932,-177.103,8.652,148.870
C09660=1136.479,295.198,-73.963,-177.100,8.656,148.870
C09661=1136.474,295.446,-73.994,-177.097,8.659,148.870
C09662=1136.471,295.694,-74.024,-177.095,8.662,148.870
C09663=1136.466,295.942,-74.055,-177.092,8.666,148.870
C09664=1136.462,296.190,-74.087,-177.089,8.669,148.870
C09665=1136.458,296.438,-74.118,-177.086,8.673,148.870
C09666=1136.453,296.686,-74.149,-177.084,8.676,148.871
C09667=1136.450,296.935,-74.179,-177.081,8.679,148.871
C09668=1136.445,297.182,-74.210,-177.078,8.683,148.871
C09669=1136.442,297.430,-74.242,-177.076,8.686,148.871
C09670=1136.437,297.678,-74.272,-177.073,8.689,148.871
C09671=1136.432,297.926,-74.303,-177.070,8.693,148.871
C09672=1136.428,298.175,-74.334,-177.068,8.697,148.871
C09673=1136.424,298.422,-74.366,-177.065,8.700,148.871
C09674=1136.421,298.671,-74.396,-177.062,8.704,148.871
C09675=1136.416,298.919,-74.427,-177.060,8.707,148.872
C09676=1136.413,299.167,-74.459,-177.057,8.711,148.872
C09677=1136.408,299.415,-74.490,-177.054,8.714,148.872
C09678=1136.403,299.663,-74.520,-177.051,8.718,148.872
C09679=1136.400,299.911,-74.552,-177.049,8.721,148.872
C09680=1136.395,300.159,-74.583,-177.047,8.724,148.872
C09681=1136.391,300.407,-74.615,-177.043,8.728,148.872
C09682=1136.387,300.655,-74.646,-177.041,8.731,148.873
C09683=1136.383,300.903,-74.678,-177.038,8.735,148.873
C09684=1136.378,301.151,-74.708,-177.036,8.739,148.873
C09685=1136.374,301.399,-74.739,-177.032,8.742,148.873
C09686=1136.370,301.647,-74.771,-177.030,8.746,148.873
C09687=1136.366,301.895,-74.802,-177.028,8.749,148.873
C09688=1136.362,302.143,-74.834,-177.025,8.753,148.873
C09689=1136.358,302.391,-74.865,-177.022,8.756,148.873
C09690=1136.353,302.639,-74.896,-177.019,8.760,148.874
C09691=1136.350,302.887,-74.928,-177.017,8.763,148.874
C09692=1136.345,303.135,-74.959,-177.014,8.767,148.874
C09693=1136.341,303.383,-74.991,-177.011,8.770,148.874
C09694=1136.337,303.631,-75.021,-177.008,8.774,148.874
C09695=1136.333,303.879,-75.053,-177.006,8.778,148.874
C09696=1136.329,304.126,-75.085,-177.003,8.781,148.875
C09697=1136.325,304.375,-75.116,-177.000,8.785,148.875
C09698=1136.321,304.623,-75.148,-176.997,8.788,148.875
C09699=1136.316,304.870,-75.180,-176.995,8.792,148.875
C09700=1136.312,305.119,-75.211,-176.992,8.795,148.875
C09701=1136.308,305.366,-75.242,-176.990,8.798,148.875
C09702=1136.304,305.614,-75.274,-176.987,8.803,148.876
C09703=1136.286,306.680,-75.412,-177.856,10.498,149.535
C09704=1136.282,306.928,-75.444,-177.853,10.501,149.535
C09705=1136.278,307.176,-75.477,-177.850,10.503,149.535
C09706=1136.273,307.423,-75.508,-177.847,10.506,149.534
C09707=1136.270,307.671,-75.541,-177.844,10.509,149.534
C09708=1136.266,307.923,-75.574,-177.841,10.511,149.534
C09709=1136.261,308.174,-75.606,-177.837,10.513,149.534
C09710=1136.257,308.426,-75.639,-177.834,10.516,149.534
C09711=1136.253,308.678,-75.671,-177.831,10.519,149.533
C09712=1136.249,308.925,-75.703,-177.828,10.521,149.533
C09713=1136.245,309.173,-75.736,-177.825,10.524,149.533
C09714=1136.241,309.421,-75.767,-177.821,10.526,149.533
C09715=1136.236,309.669,-75.800,-177.819,10.529,149.533
C09716=1136.232,309.917,-75.832,-177.815,10.531,149.532
C09717=1136.228,310.165,-75.865,-177.812,10.534,149.532
C09718=1136.225,310.413,-75.897,-177.809,10.537,149.532
C09719=1136.220,310.660,-75.929,-177.806,10.539,149.532
C09720=1136.216,310.908,-75.961,-177.803,10.542,149.532
C09721=1136.212,311.156,-75.994,-177.799,10.544,149.531
C09722=1136.208,311.404,-76.026,-177.796,10.547,149.531
C09723=1136.204,311.652,-76.059,-177.793,10.550,149.531
C09724=1136.200,311.900,-76.091,-177.790,10.552,149.531
C09725=1136.195,312.148,-76.123,-177.787,10.555,149.531
C09726=1136.192,312.395,-76.155,-177.783,10.557,149.530
C09727=1136.187,312.643,-76.188,-177.781,10.560,149.530
C09728=1136.184,312.891,-76.220,-177.778,10.562,149.530
C09729=1136.179,313.139,-76.253,-177.775,10.564,149.530
C09730=1136.176,313.387,-76.285,-177.772,10.567,149.530
C09731=1136.172,313.635,-76.318,-177.768,10.569,149.530
C09732=1136.167,313.883,-76.350,-177.765,10.572,149.529
C09733=1136.163,314.130,-76.382,-177.762,10.574,149.529
C09734=1136.159,314.378,-76.415,-177.759,10.577,149.529
C09735=1136.155,314.626,-76.447,-177.756,10.580,149.529
C09736=1136.151,314.874,-76.480,-177.752,10.582,149.529
C09737=1136.147,315.122,-76.513,-177.749,10.585,149.529
C09738=1136.143,315.369,-76.545,-177.746,10.587,149.528
C09739=1136.139,315.618,-76.578,-177.743,10.590,149.528
C09740=1136.135,315.865,-76.611,-177.740,10.593,149.528
C09741=1136.131,316.113,-76.643,-177.737,10.595,149.528
C09742=1136.127,316.361,-76.676,-177.733,10.597,149.527
C09743=1136.123,316.609,-76.709,-177.730,10.600,149.527
C09744=1136.119,316.857,-76.741,-177.727,10.603,149.527
C09745=1136.115,317.105,-76.774,-177.724,10.605,149.527
C09746=1136.110,317.352,-76.807,-177.721,10.608,149.527
C09747=1136.106,317.600,-76.839,-177.717,10.610,149.527
C09748=1136.102,317.847,-76.872,-177.714,10.613,149.526
C09749=1136.098,318.095,-76.905,-177.711,10.615,149.526
C09750=1136.094,318.344,-76.938,-177.708,10.618,149.526
C09751=1136.090,318.591,-76.971,-177.705,10.621,149.526
C09752=1136.086,318.839,-77.003,-177.702,10.622,149.526
C09753=1136.082,319.086,-77.036,-177.699,10.625,149.525
C09754=1136.078,319.334,-77.070,-177.696,10.628,149.525
C09755=1136.073,319.582,-77.102,-177.693,10.630,149.525
C09756=1136.069,319.830,-77.135,-177.689,10.632,149.525
C09757=1136.066,320.078,-77.168,-177.686,10.635,149.525
C09758=1136.062,320.325,-77.201,-177.683,10.638,149.524
C09759=1136.058,320.574,-77.234,-177.680,10.640,149.524
C09760=1136.054,320.787,-77.263,-177.677,10.643,149.524
C09761=1136.051,321.001,-77.291,-177.674,10.645,149.524
C09762=1136.048,321.214,-77.320,-177.672,10.647,149.524
C09763=1136.044,321.428,-77.348,-177.669,10.649,149.524
C09764=1136.040,321.641,-77.376,-177.666,10.651,149.523
C09765=1136.038,321.855,-77.405,-177.663,10.654,149.523
C09766=1136.034,322.068,-77.433,-177.661,10.655,149.523
C09767=1136.030,322.282,-77.461,-177.658,10.658,149.523
C09768=1136.026,322.529,-77.495,-177.654,10.661,149.523
C09769=1136.022,322.777,-77.528,-177.651,10.663,149.523
C09770=1136.018,323.026,-77.561,-177.649,10.665,149.522
C09771=1136.014,323.273,-77.594,-177.645,10.667,149.522
C09772=1136.010,323.521,-77.628,-177.642,10.670,149.522
C09773=1136.006,323.769,-77.661,-177.639,10.673,149.522
C09774=1136.002,324.016,-77.695,-177.636,10.675,149.522
C09775=1135.998,324.264,-77.728,-177.633,10.678,149.522
C09776=1135.994,324.511,-77.761,-177.630,10.680,149.521
C09777=1135.990,324.759,-77.794,-177.626,10.683,149.521
C09778=1135.986,325.007,-77.827,-177.623,10.685,149.521
C09779=1135.982,325.255,-77.861,-177.620,10.688,149.521
C09780=1135.978,325.503,-77.894,-177.617,10.690,149.520
C09781=1135.974,325.751,-77.927,-177.613,10.693,149.520
C09782=1135.970,325.998,-77.961,-177.610,10.696,149.520
C09783=1135.966,326.246,-77.994,-177.607,10.698,149.520
C09784=1135.962,326.493,-78.027,-177.604,10.701,149.520
C09785=1135.958,326.742,-78.061,-177.601,10.703,149.520
C09786=1135.954,326.989,-78.094,-177.598,10.706,149.519
C09787=1135.950,327.237,-78.128,-177.594,10.708,149.519
C09788=1135.946,327.484,-78.161,-177.591,10.711,149.519
C09789=1135.942,327.732,-78.194,-177.588,10.713,149.519
C09790=1135.938,327.979,-78.228,-177.585,10.716,149.519
C09791=1135.934,328.228,-78.262,-177.581,10.718,149.518
C09792=1135.930,328.476,-78.295,-177.578,10.721,149.518
C09793=1135.925,328.723,-78.328,-177.575,10.724,149.518
C09794=1135.922,328.970,-78.362,-177.572,10.726,149.518
C09795=1135.918,329.218,-78.395,-177.568,10.728,149.518
C09796=1135.914,329.466,-78.430,-177.565,10.731,149.517
C09797=1135.910,329.714,-78.463,-177.562,10.734,149.517
C09798=1135.905,329.962,-78.497,-177.559,10.736,149.517
C09799=1135.901,330.209,-78.530,-177.556,10.739,149.517
C09800=1135.898,330.457,-78.564,-177.553,10.741,149.517
C09801=1135.894,330.704,-78.598,-177.549,10.744,149.516
C09802=1135.890,330.952,-78.631,-177.546,10.746,149.516
C09803=1135.885,331.200,-78.665,-177.543,10.749,149.516
C09804=1135.882,331.448,-78.699,-177.540,10.751,149.516
C09805=1135.878,331.695,-78.733,-177.537,10.753,149.516
C09806=1135.874,331.943,-78.766,-177.534,10.756,149.515
C09807=1135.869,332.190,-78.800,-177.530,10.758,149.515
C09808=1135.866,332.439,-78.834,-177.527,10.761,149.515
C09809=1135.862,332.686,-78.868,-177.524,10.763,149.515
C09810=1135.858,332.933,-78.901,-177.521,10.766,149.515
C09811=1135.854,333.182,-78.936,-177.517,10.768,149.514
C09812=1135.850,333.429,-78.970,-177.515,10.771,149.514
C09813=1135.846,333.676,-79.003,-177.511,10.773,149.514
C09814=1135.842,333.925,-79.038,-177.508,10.776,149.514
C09815=1135.838,334.172,-79.072,-177.505,10.778,149.514
C09816=1135.835,334.385,-79.100,-177.502,10.781,149.513
C09817=1135.831,334.598,-79.130,-177.499,10.783,149.513
C09818=1135.828,334.812,-79.160,-177.496,10.786,149.513
C09819=1135.824,335.025,-79.188,-177.493,10.787,149.513
C09820=1135.821,335.239,-79.218,-177.491,10.789,149.513
C09821=1135.817,335.452,-79.247,-177.488,10.792,149.513
C09822=1135.814,335.665,-79.276,-177.485,10.794,149.512
C09823=1135.810,335.879,-79.306,-177.482,10.796,149.512
C09824=1135.807,336.126,-79.340,-177.479,10.799,149.512
C09825=1135.803,336.374,-79.373,-177.476,10.801,149.512
C09826=1135.799,336.622,-79.408,-177.473,10.804,149.512
C09827=1135.795,336.869,-79.442,-177.469,10.806,149.511
C09828=1135.790,337.117,-79.476,-177.466,10.809,149.511
C09829=1135.787,337.365,-79.511,-177.463,10.811,149.511
C09830=1135.782,337.613,-79.544,-177.460,10.814,149.511
C09831=1135.779,337.860,-79.579,-177.456,10.816,149.511
C09832=1135.774,338.108,-79.613,-177.453,10.819,149.510
C09833=1135.771,338.355,-79.647,-177.450,10.821,149.510
C09834=1135.767,338.603,-79.682,-177.447,10.823,149.510
C09835=1135.763,338.850,-79.716,-177.444,10.826,149.510
C09836=1135.759,339.098,-79.751,-177.441,10.828,149.510
C09837=1135.755,339.345,-79.784,-177.438,10.831,149.509
C09838=1135.751,339.593,-79.819,-177.434,10.833,149.509
C09839=1135.747,339.841,-79.853,-177.431,10.836,149.509
C09840=1135.743,340.088,-79.888,-177.428,10.838,149.509
C09841=1135.739,340.336,-79.922,-177.425,10.841,149.509
C09842=1135.735,340.583,-79.956,-177.421,10.843,149.508
C09843=1135.731,340.831,-79.991,-177.418,10.846,149.508
C09844=1135.727,341.078,-80.025,-177.415,10.848,149.508
C09845=1135.723,341.327,-80.060,-177.411,10.851,149.508
C09846=1135.719,341.574,-80.094,-177.408,10.853,149.507
C09847=1135.715,341.822,-80.129,-177.405,10.856,149.507
C09848=1135.711,342.069,-80.163,-177.402,10.858,149.507
C09849=1135.707,342.317,-80.197,-177.399,10.861,149.507
C09850=1135.703,342.564,-80.232,-177.395,10.863,149.507
C09851=1135.699,342.812,-80.267,-177.392,10.866,149.506
C09852=1135.695,343.059,-80.301,-177.389,10.868,149.506
C09853=1135.691,343.307,-80.336,-177.386,10.871,149.506
C09854=1135.687,343.555,-80.370,-177.382,10.873,149.506
C09855=1135.684,343.802,-80.405,-177.379,10.876,149.506
C09856=1135.679,344.049,-80.440,-177.376,10.878,149.506
C09857=1135.675,344.297,-80.475,-177.372,10.881,149.505
C09858=1135.672,344.544,-80.509,-177.369,10.883,149.505
C09859=1135.668,344.792,-80.544,-177.366,10.886,149.505
C09860=1135.664,345.040,-80.579,-177.363,10.888,149.505
C09861=1135.659,345.287,-80.613,-177.360,10.891,149.505
C09862=1135.656,345.535,-80.648,-177.356,10.893,149.504
C09863=1135.652,345.782,-80.683,-177.353,10.896,149.504
C09864=1135.648,346.030,-80.718,-177.350,10.898,149.504
C09865=1135.644,346.277,-80.753,-177.346,10.901,149.504
C09866=1135.640,346.525,-80.787,-177.343,10.903,149.503
C09867=1135.636,346.773,-80.822,-177.340,10.906,149.503
C09868=1135.632,347.020,-80.857,-177.337,10.908,149.503
C09869=1135.628,347.268,-80.892,-177.333,10.911,149.503
C09870=1135.624,347.515,-80.927,-177.330,10.913,149.503
C09871=1135.621,347.762,-80.961,-177.327,10.916,149.502
C09872=1135.617,347.976,-80.992,-177.324,10.917,149.502
C09873=1135.614,348.190,-81.022,-177.321,10.920,149.502
C09874=1135.610,348.402,-81.052,-177.319,10.922,149.502
C09875=1135.607,348.615,-81.082,-177.315,10.924,149.502
C09876=1135.604,348.828,-81.112,-177.313,10.926,149.502
C09877=1135.600,349.042,-81.142,-177.310,10.929,149.501
C09878=1135.597,349.256,-81.173,-177.307,10.931,149.501
C09879=1135.593,349.468,-81.203,-177.305,10.933,149.501
C09880=1135.590,349.716,-81.237,-177.301,10.936,149.501
C09881=1135.586,349.964,-81.273,-177.297,10.938,149.500
C09882=1135.582,350.210,-81.308,-177.293,10.941,149.500
C09883=1135.578,350.458,-81.343,-177.289,10.944,149.500
C09884=1135.574,350.706,-81.378,-177.285,10.947,149.500
C09885=1135.570,350.954,-81.413,-177.281,10.950,149.499
C09886=1135.566,351.201,-81.448,-177.278,10.952,149.499
C09887=1135.562,351.448,-81.484,-177.274,10.954,149.499
C09888=1135.558,351.696,-81.519,-177.270,10.958,149.499
C09889=1135.554,351.943,-81.554,-177.267,10.960,149.498
C09890=1135.550,352.191,-81.590,-177.263,10.963,149.498
C09891=1135.547,352.438,-81.625,-177.260,10.965,149.498
C09892=1135.543,352.686,-81.661,-177.256,10.969,149.498
C09893=1135.538,352.933,-81.695,-177.252,10.971,149.497
C09894=1135.535,353.181,-81.731,-177.249,10.973,149.497
C09895=1135.531,353.428,-81.766,-177.245,10.977,149.497
C09896=1135.527,353.676,-81.802,-177.241,10.979,149.496
C09897=1135.523,353.923,-81.837,-177.238,10.981,149.496
C09898=1135.519,354.170,-81.872,-177.234,10.984,149.496
C09899=1135.515,354.418,-81.907,-177.230,10.986,149.495
C09900=1135.512,354.666,-81.943,-177.227,10.989,149.495
C09901=1135.508,354.913,-81.978,-177.223,10.992,149.495
C09902=1135.503,355.160,-82.014,-177.219,10.994,149.495
C09903=1135.499,355.408,-82.050,-177.216,10.997,149.494
C09904=1135.496,355.655,-82.085,-177.212,11.000,149.494
C09905=1135.492,355.903,-82.121,-177.208,11.002,149.494
C09906=1135.488,356.150,-82.156,-177.205,11.005,149.494
C09907=1135.485,356.398,-82.192,-177.201,11.007,149.493
C09908=1135.481,356.645,-82.227,-177.197,11.010,149.493
C09909=1135.477,356.892,-82.263,-177.194,11.012,149.493
C09910=1135.472,357.140,-82.299,-177.190,11.015,149.493
C09911=1135.469,357.387,-82.334,-177.187,11.017,149.492
C09912=1135.465,357.635,-82.370,-177.183,11.020,149.492
C09913=1135.462,357.882,-82.406,-177.180,11.022,149.492
C09914=1135.458,358.129,-82.442,-177.176,11.025,149.491
C09915=1135.453,358.376,-82.477,-177.173,11.027,149.491
C09916=1135.449,358.624,-82.513,-177.169,11.030,149.491
C09917=1135.446,358.871,-82.549,-177.166,11.032,149.491
C09918=1135.442,359.119,-82.584,-177.162,11.034,149.490
C09919=1135.438,359.366,-82.621,-177.159,11.037,149.490
C09920=1135.434,359.614,-82.656,-177.156,11.039,149.490
C09921=1135.431,359.861,-82.692,-177.152,11.042,149.490
C09922=1135.427,360.109,-82.728,-177.149,11.044,149.489
C09923=1135.423,360.356,-82.764,-177.145,11.046,149.489
C09924=1135.419,360.603,-82.800,-177.141,11.050,149.489
C09925=1135.416,360.851,-82.836,-177.138,11.052,149.488
C09926=1135.411,361.099,-82.872,-177.134,11.054,149.488
C09927=1135.408,361.345,-82.908,-177.131,11.057,149.488
C09928=1135.405,361.559,-82.939,-177.128,11.058,149.488
C09929=1135.401,361.771,-82.970,-177.125,11.061,149.488
C09930=1135.398,361.985,-83.000,-177.122,11.063,149.487
C09931=1135.394,362.198,-83.032,-177.120,11.064,149.487
C09932=1135.391,362.411,-83.063,-177.116,11.067,149.487
C09933=1135.388,362.624,-83.094,-177.114,11.069,149.487
C09934=1135.385,362.837,-83.125,-177.111,11.071,149.487
C09935=1135.382,363.050,-83.156,-177.108,11.073,149.486
C09936=1135.377,363.297,-83.192,-177.105,11.075,149.486
C09937=1135.374,363.544,-83.228,-177.101,11.078,149.486
C09938=1135.369,363.792,-83.264,-177.098,11.080,149.485
C09939=1135.366,364.040,-83.300,-177.095,11.083,149.485
C09940=1135.362,364.286,-83.336,-177.091,11.085,149.485
C09941=1135.358,364.534,-83.372,-177.089,11.087,149.485
C09942=1135.355,364.781,-83.409,-177.085,11.089,149.485
C09943=1135.350,365.028,-83.446,-177.082,11.092,149.484
C09944=1135.347,365.276,-83.481,-177.078,11.094,149.484
C09945=1135.343,365.523,-83.518,-177.075,11.096,149.484
C09946=1135.339,365.770,-83.553,-177.072,11.099,149.483
C09947=1135.335,366.018,-83.590,-177.068,11.101,149.483
C09948=1135.331,366.265,-83.626,-177.066,11.103,149.483
C09949=1135.328,366.513,-83.663,-177.062,11.105,149.483
C09950=1135.324,366.760,-83.699,-177.059,11.108,149.483
C09951=1135.320,367.008,-83.736,-177.056,11.110,149.482
C09952=1135.317,367.255,-83.772,-177.052,11.113,149.482
C09953=1135.313,367.502,-83.809,-177.050,11.114,149.482
C09954=1135.308,367.750,-83.845,-177.046,11.117,149.482
C09955=1135.305,367.997,-83.881,-177.043,11.119,149.482
C09956=1135.301,368.244,-83.918,-177.040,11.122,149.481
C09957=1135.297,368.491,-83.954,-177.037,11.124,149.481
C09958=1135.293,368.738,-83.990,-177.034,11.126,149.481
C09959=1135.289,368.986,-84.027,-177.031,11.129,149.481
C09960=1135.286,369.233,-84.064,-177.027,11.131,149.480
C09961=1135.282,369.480,-84.101,-177.025,11.133,149.480
C09962=1135.279,369.727,-84.137,-177.021,11.135,149.480
C09963=1135.274,369.975,-84.173,-177.018,11.138,149.480
C09964=1135.270,370.222,-84.210,-177.015,11.139,149.479
C09965=1135.267,370.469,-84.246,-177.012,11.142,149.479
C09966=1135.263,370.716,-84.283,-177.009,11.144,149.479
C09967=1135.259,370.963,-84.320,-177.006,11.146,149.479
C09968=1135.256,371.211,-84.357,-177.003,11.149,149.479
C09969=1135.252,371.458,-84.393,-177.000,11.151,149.479
C09970=1135.247,371.706,-84.430,-176.997,11.153,149.478
C09971=1135.244,371.953,-84.466,-176.994,11.155,149.478
C09972=1135.240,372.200,-84.503,-176.991,11.158,149.478
C09973=1135.236,372.448,-84.540,-176.988,11.160,149.478
C09974=1135.232,372.695,-84.577,-176.985,11.162,149.478
C09975=1135.229,372.942,-84.613,-176.982,11.164,149.477
C09976=1135.225,373.189,-84.650,-176.979,11.167,149.477
C09977=1135.221,373.436,-84.687,-176.977,11.169,149.477
C09978=1135.217,373.684,-84.724,-176.973,11.171,149.477
C09979=1135.214,373.931,-84.760,-176.970,11.174,149.477
C09980=1135.210,374.178,-84.797,-176.968,11.176,149.477
C09981=1135.206,374.426,-84.834,-176.965,11.178,149.476
C09982=1135.202,374.672,-84.871,-176.962,11.180,149.476
C09983=1135.199,374.920,-84.908,-176.959,11.183,149.476
C09984=1135.195,375.133,-84.940,-176.956,11.184,149.476
C09985=1135.192,375.346,-84.972,-176.954,11.186,149.476
C09986=1135.189,375.558,-85.003,-176.952,11.188,149.476
C09987=1135.185,375.772,-85.035,-176.949,11.190,149.476
C09988=1135.182,375.985,-85.067,-176.947,11.192,149.476
C09989=1135.179,376.197,-85.099,-176.945,11.194,149.475
C09990=1135.176,376.410,-85.131,-176.942,11.196,149.475
C09991=1135.173,376.623,-85.163,-176.940,11.198,149.475
C09992=1135.169,376.871,-85.200,-176.937,11.199,149.475
C09993=1135.165,377.118,-85.236,-176.934,11.202,149.475
C09994=1135.161,377.365,-85.274,-176.931,11.204,149.475
C09995=1135.158,377.612,-85.311,-176.928,11.207,149.475
C09996=1135.154,377.859,-85.348,-176.926,11.209,149.475
//INST
///DATE 2021/06/25 14:31
///ATTR SC,RW,RJ
////FRAME ROBOT
///GROUP1 RB1
NOP
MOVL C00000 V=800.0 PL=0
MOVL C00001 V=800.0 PL=0
MOVL C00002 V=800.0 PL=0
MOVL C00003 V=800.0 PL=0
MOVL C00004 V=800.0 PL=0
MOVL C00005 V=800.0 PL=0
MOVL C00006 V=800.0 PL=0
MOVL C00007 V=800.0 PL=0
MOVL C00008 V=800.0 PL=0
MOVL C00009 V=800.0 PL=0
MOVL C00010 V=800.0 PL=0
MOVL C00011 V=800.0 PL=0
MOVL C00012 V=800.0 PL=0
MOVL C00013 V=800.0 PL=0
MOVL C00014 V=800.0 PL=0
MOVL C00015 V=800.0 PL=0
MOVL C00016 V=800.0 PL=0
MOVL C00017 V=800.0 PL=0
MOVL C00018 V=800.0 PL=0
MOVL C00019 V=800.0 PL=0
MOVL C00020 V=800.0 PL=0
MOVL C00021 V=800.0 PL=0
MOVL C00022 V=800.0 PL=0
MOVL C00023 V=800.0 PL=0
MOVL C00024 V=800.0 PL=0
MOVL C00025 V=800.0 PL=0
MOVL C00026 V=800.0 PL=0
MOVL C00027 V=800.0 PL=0
MOVL C00028 V=800.0 PL=0
MOVL C00029 V=800.0 PL=0
MOVL C00030 V=800.0 PL=0
MOVL C00031 V=800.0 PL=0
MOVL C00032 V=800.0 PL=0
MOVL C00033 V=800.0 PL=0
MOVL C00034 V=800.0 PL=0
MOVL C00035 V=800.0 PL=0
MOVL C00036 V=800.0 PL=0
MOVL C00037 V=800.0 PL=0
MOVL C00038 V=800.0 PL=0
MOVL C00039 V=800.0 PL=0
MOVL C00040 V=800.0 PL=0
MOVL C00041 V=800.0 PL=0
MOVL C00042 V=800.0 PL=0
MOVL C00043 V=800.0 PL=0
MOVL C00044 V=800.0 PL=0
MOVL C00045 V=800.0 PL=0
MOVL C00046 V=800.0 PL=0
MOVL C00047 V=800.0 PL=0
MOVL C00048 V=800.0 PL=0
MOVL C00049 V=800.0 PL=0
MOVL C00050 V=800.0 PL=0
MOVL C00051 V=800.0 PL=0
MOVL C00052 V=800.0 PL=0
MOVL C00053 V=800.0 PL=0
MOVL C00054 V=800.0 PL=0
MOVL C00055 V=800.0 PL=0
MOVL C00056 V=800.0 PL=0
MOVL C00057 V=800.0 PL=0
MOVL C00058 V=800.0 PL=0
MOVL C00059 V=800.0 PL=0
MOVL C00060 V=800.0 PL=0
MOVL C00061 V=800.0 PL=0
MOVL C00062 V=800.0 PL=0
MOVL C00063 V=800.0 PL=0
MOVL C00064 V=800.0 PL=0
MOVL C00065 V=800.0 PL=0
MOVL C00066 V=800.0 PL=0
MOVL C00067 V=800.0 PL=0
MOVL C00068 V=800.0 PL=0
MOVL C00069 V=800.0 PL=0
MOVL C00070 V=800.0 PL=0
MOVL C00071 V=800.0 PL=0
MOVL C00072 V=800.0 PL=0
MOVL C00073 V=800.0 PL=0
MOVL C00074 V=800.0 PL=0
MOVL C00075 V=800.0 PL=0
MOVL C00076 V=800.0 PL=0
MOVL C00077 V=800.0 PL=0
MOVL C00078 V=800.0 PL=0
MOVL C00079 V=800.0 PL=0
MOVL C00080 V=800.0 PL=0
MOVL C00081 V=800.0 PL=0
MOVL C00082 V=800.0 PL=0
MOVL C00083 V=800.0 PL=0
MOVL C00084 V=800.0 PL=0
MOVL C00085 V=800.0 PL=0
MOVL C00086 V=800.0 PL=0
MOVL C00087 V=800.0 PL=0
MOVL C00088 V=800.0 PL=0
MOVL C00089 V=800.0 PL=0
MOVL C00090 V=800.0 PL=0
MOVL C00091 V=800.0 PL=0
MOVL C00092 V=800.0 PL=0
MOVL C00093 V=800.0 PL=0
MOVL C00094 V=800.0 PL=0
MOVL C00095 V=800.0 PL=0
MOVL C00096 V=800.0 PL=0
MOVL C00097 V=800.0 PL=0
MOVL C00098 V=800.0 PL=0
MOVL C00099 V=800.0 PL=0
MOVL C00100 V=800.0 PL=0
MOVL C00101 V=800.0 PL=0
MOVL C00102 V=800.0 PL=0
MOVL C00103 V=800.0 PL=0
MOVL C00104 V=800.0 PL=0
MOVL C00105 V=800.0 PL=0
MOVL C00106 V=800.0 PL=0
MOVL C00107 V=800.0 PL=0
MOVL C00108 V=800.0 PL=0
MOVL C00109 V=800.0 PL=0
MOVL C00110 V=800.0 PL=0
MOVL C00111 V=800.0 PL=0
MOVL C00112 V=800.0 PL=0
MOVL C00113 V=800.0 PL=0
MOVL C00114 V=800.0 PL=0
MOVL C00115 V=800.0 PL=0
MOVL C00116 V=800.0 PL=0
MOVL C00117 V=800.0 PL=0
MOVL C00118 V=800.0 PL=0
MOVL C00119 V=800.0 PL=0
MOVL C00120 V=800.0 PL=0
MOVL C00121 V=800.0 PL=0
MOVL C00122 V=800.0 PL=0
MOVL C00123 V=800.0 PL=0
MOVL C00124 V=800.0 PL=0
MOVL C00125 V=800.0 PL=0
MOVL C00126 V=800.0 PL=0
MOVL C00127 V=800.0 PL=0
MOVL C00128 V=800.0 PL=0
MOVL C00129 V=800.0 PL=0
MOVL C00130 V=800.0 PL=0
MOVL C00131 V=800.0 PL=0
MOVL C00132 V=800.0 PL=0
MOVL C00133 V=800.0 PL=0
MOVL C00134 V=800.0 PL=0
MOVL C00135 V=800.0 PL=0
MOVL C00136 V=800.0 PL=0
MOVL C00137 V=800.0 PL=0
MOVL C00138 V=800.0 PL=0
MOVL C00139 V=800.0 PL=0
MOVL C00140 V=800.0 PL=0
MOVL C00141 V=800.0 PL=0
MOVL C00142 V=800.0 PL=0
MOVL C00143 V=800.0 PL=0
MOVL C00144 V=800.0 PL=0
MOVL C00145 V=800.0 PL=0
MOVL C00146 V=800.0 PL=0
MOVL C00147 V=800.0 PL=0
MOVL C00148 V=800.0 PL=0
MOVL C00149 V=800.0 PL=0
MOVL C00150 V=800.0 PL=0
MOVL C00151 V=800.0 PL=0
MOVL C00152 V=800.0 PL=0
MOVL C00153 V=800.0 PL=0
MOVL C00154 V=800.0 PL=0
MOVL C00155 V=800.0 PL=0
MOVL C00156 V=800.0 PL=0
MOVL C00157 V=800.0 PL=0
MOVL C00158 V=800.0 PL=0
MOVL C00159 V=800.0 PL=0
MOVL C00160 V=800.0 PL=0
MOVL C00161 V=800.0 PL=0
MOVL C00162 V=800.0 PL=0
MOVL C00163 V=800.0 PL=0
MOVL C00164 V=800.0 PL=0
MOVL C00165 V=800.0 PL=0
MOVL C00166 V=800.0 PL=0
MOVL C00167 V=800.0 PL=0
MOVL C00168 V=800.0 PL=0
MOVL C00169 V=800.0 PL=0
MOVL C00170 V=800.0 PL=0
MOVL C00171 V=800.0 PL=0
MOVL C00172 V=800.0 PL=0
MOVL C00173 V=800.0 PL=0
MOVL C00174 V=800.0 PL=0
MOVL C00175 V=800.0 PL=0
MOVL C00176 V=800.0 PL=0
MOVL C00177 V=800.0 PL=0
MOVL C00178 V=800.0 PL=0
MOVL C00179 V=800.0 PL=0
MOVL C00180 V=800.0 PL=0
MOVL C00181 V=800.0 PL=0
MOVL C00182 V=800.0 PL=0
MOVL C00183 V=800.0 PL=0
MOVL C00184 V=800.0 PL=0
MOVL C00185 V=800.0 PL=0
MOVL C00186 V=800.0 PL=0
MOVL C00187 V=800.0 PL=0
MOVL C00188 V=800.0 PL=0
MOVL C00189 V=800.0 PL=0
MOVL C00190 V=800.0 PL=0
MOVL C00191 V=800.0 PL=0
MOVL C00192 V=800.0 PL=0
MOVL C00193 V=800.0 PL=0
MOVL C00194 V=800.0 PL=0
MOVL C00195 V=800.0 PL=0
MOVL C00196 V=800.0 PL=0
MOVL C00197 V=800.0 PL=0
MOVL C00198 V=800.0 PL=0
MOVL C00199 V=800.0 PL=0
MOVL C00200 V=800.0 PL=0
MOVL C00201 V=800.0 PL=0
MOVL C00202 V=800.0 PL=0
MOVL C00203 V=800.0 PL=0
MOVL C00204 V=800.0 PL=0
MOVL C00205 V=800.0 PL=0
MOVL C00206 V=800.0 PL=0
MOVL C00207 V=800.0 PL=0
MOVL C00208 V=800.0 PL=0
MOVL C00209 V=800.0 PL=0
MOVL C00210 V=800.0 PL=0
MOVL C00211 V=800.0 PL=0
MOVL C00212 V=800.0 PL=0
MOVL C00213 V=800.0 PL=0
MOVL C00214 V=800.0 PL=0
MOVL C00215 V=800.0 PL=0
MOVL C00216 V=800.0 PL=0
MOVL C00217 V=800.0 PL=0
MOVL C00218 V=800.0 PL=0
MOVL C00219 V=800.0 PL=0
MOVL C00220 V=800.0 PL=0
MOVL C00221 V=800.0 PL=0
MOVL C00222 V=800.0 PL=0
MOVL C00223 V=800.0 PL=0
MOVL C00224 V=800.0 PL=0
MOVL C00225 V=800.0 PL=0
MOVL C00226 V=800.0 PL=0
MOVL C00227 V=800.0 PL=0
MOVL C00228 V=800.0 PL=0
MOVL C00229 V=800.0 PL=0
MOVL C00230 V=800.0 PL=0
MOVL C00231 V=800.0 PL=0
MOVL C00232 V=800.0 PL=0
MOVL C00233 V=800.0 PL=0
MOVL C00234 V=800.0 PL=0
MOVL C00235 V=800.0 PL=0
MOVL C00236 V=800.0 PL=0
MOVL C00237 V=800.0 PL=0
MOVL C00238 V=800.0 PL=0
MOVL C00239 V=800.0 PL=0
MOVL C00240 V=800.0 PL=0
MOVL C00241 V=800.0 PL=0
MOVL C00242 V=800.0 PL=0
MOVL C00243 V=800.0 PL=0
MOVL C00244 V=800.0 PL=0
MOVL C00245 V=800.0 PL=0
MOVL C00246 V=800.0 PL=0
MOVL C00247 V=800.0 PL=0
MOVL C00248 V=800.0 PL=0
MOVL C00249 V=800.0 PL=0
MOVL C00250 V=800.0 PL=0
MOVL C00251 V=800.0 PL=0
MOVL C00252 V=800.0 PL=0
MOVL C00253 V=800.0 PL=0
MOVL C00254 V=800.0 PL=0
MOVL C00255 V=800.0 PL=0
MOVL C00256 V=800.0 PL=0
MOVL C00257 V=800.0 PL=0
MOVL C00258 V=800.0 PL=0
MOVL C00259 V=800.0 PL=0
MOVL C00260 V=800.0 PL=0
MOVL C00261 V=800.0 PL=0
MOVL C00262 V=800.0 PL=0
MOVL C00263 V=800.0 PL=0
MOVL C00264 V=800.0 PL=0
MOVL C00265 V=800.0 PL=0
MOVL C00266 V=800.0 PL=0
MOVL C00267 V=800.0 PL=0
MOVL C00268 V=800.0 PL=0
MOVL C00269 V=800.0 PL=0
MOVL C00270 V=800.0 PL=0
MOVL C00271 V=800.0 PL=0
MOVL C00272 V=800.0 PL=0
MOVL C00273 V=800.0 PL=0
MOVL C00274 V=800.0 PL=0
MOVL C00275 V=800.0 PL=0
MOVL C00276 V=800.0 PL=0
MOVL C00277 V=800.0 PL=0
MOVL C00278 V=800.0 PL=0
MOVL C00279 V=800.0 PL=0
MOVL C00280 V=800.0 PL=0
MOVL C00281 V=800.0 PL=0
MOVL C00282 V=800.0 PL=0
MOVL C00283 V=800.0 PL=0
MOVL C00284 V=800.0 PL=0
MOVL C00285 V=800.0 PL=0
MOVL C00286 V=800.0 PL=0
MOVL C00287 V=800.0 PL=0
MOVL C00288 V=800.0 PL=0
MOVL C00289 V=800.0 PL=0
MOVL C00290 V=800.0 PL=0
MOVL C00291 V=800.0 PL=0
MOVL C00292 V=800.0 PL=0
MOVL C00293 V=800.0 PL=0
MOVL C00294 V=800.0 PL=0
MOVL C00295 V=800.0 PL=0
MOVL C00296 V=800.0 PL=0
MOVL C00297 V=800.0 PL=0
MOVL C00298 V=800.0 PL=0
MOVL C00299 V=800.0 PL=0
MOVL C00300 V=800.0 PL=0
MOVL C00301 V=800.0 PL=0
MOVL C00302 V=800.0 PL=0
MOVL C00303 V=800.0 PL=0
MOVL C00304 V=800.0 PL=0
MOVL C00305 V=800.0 PL=0
MOVL C00306 V=800.0 PL=0
MOVL C00307 V=800.0 PL=0
MOVL C00308 V=800.0 PL=0
MOVL C00309 V=800.0 PL=0
MOVL C00310 V=800.0 PL=0
MOVL C00311 V=800.0 PL=0
MOVL C00312 V=800.0 PL=0
MOVL C00313 V=800.0 PL=0
MOVL C00314 V=800.0 PL=0
MOVL C00315 V=800.0 PL=0
MOVL C00316 V=800.0 PL=0
MOVL C00317 V=800.0 PL=0
MOVL C00318 V=800.0 PL=0
MOVL C00319 V=800.0 PL=0
MOVL C00320 V=800.0 PL=0
MOVL C00321 V=800.0 PL=0
MOVL C00322 V=800.0 PL=0
MOVL C00323 V=800.0 PL=0
MOVL C00324 V=800.0 PL=0
MOVL C00325 V=800.0 PL=0
MOVL C00326 V=800.0 PL=0
MOVL C00327 V=800.0 PL=0
MOVL C00328 V=800.0 PL=0
MOVL C00329 V=800.0 PL=0
MOVL C00330 V=800.0 PL=0
MOVL C00331 V=800.0 PL=0
MOVL C00332 V=800.0 PL=0
MOVL C00333 V=800.0 PL=0
MOVL C00334 V=800.0 PL=0
MOVL C00335 V=800.0 PL=0
MOVL C00336 V=800.0 PL=0
MOVL C00337 V=800.0 PL=0
MOVL C00338 V=800.0 PL=0
MOVL C00339 V=800.0 PL=0
MOVL C00340 V=800.0 PL=0
MOVL C00341 V=800.0 PL=0
MOVL C00342 V=800.0 PL=0
MOVL C00343 V=800.0 PL=0
MOVL C00344 V=800.0 PL=0
MOVL C00345 V=800.0 PL=0
MOVL C00346 V=800.0 PL=0
MOVL C00347 V=800.0 PL=0
MOVL C00348 V=800.0 PL=0
MOVL C00349 V=800.0 PL=0
MOVL C00350 V=800.0 PL=0
MOVL C00351 V=800.0 PL=0
MOVL C00352 V=800.0 PL=0
MOVL C00353 V=800.0 PL=0
MOVL C00354 V=800.0 PL=0
MOVL C00355 V=800.0 PL=0
MOVL C00356 V=800.0 PL=0
MOVL C00357 V=800.0 PL=0
MOVL C00358 V=800.0 PL=0
MOVL C00359 V=800.0 PL=0
MOVL C00360 V=800.0 PL=0
MOVL C00361 V=800.0 PL=0
MOVL C00362 V=800.0 PL=0
MOVL C00363 V=800.0 PL=0
MOVL C00364 V=800.0 PL=0
MOVL C00365 V=800.0 PL=0
MOVL C00366 V=800.0 PL=0
MOVL C00367 V=800.0 PL=0
MOVL C00368 V=800.0 PL=0
MOVL C00369 V=800.0 PL=0
MOVL C00370 V=800.0 PL=0
MOVL C00371 V=800.0 PL=0
MOVL C00372 V=800.0 PL=0
MOVL C00373 V=800.0 PL=0
MOVL C00374 V=800.0 PL=0
MOVL C00375 V=800.0 PL=0
MOVL C00376 V=800.0 PL=0
MOVL C00377 V=800.0 PL=0
MOVL C00378 V=800.0 PL=0
MOVL C00379 V=800.0 PL=0
MOVL C00380 V=800.0 PL=0
MOVL C00381 V=800.0 PL=0
MOVL C00382 V=800.0 PL=0
MOVL C00383 V=800.0 PL=0
MOVL C00384 V=800.0 PL=0
MOVL C00385 V=800.0 PL=0
MOVL C00386 V=800.0 PL=0
MOVL C00387 V=800.0 PL=0
MOVL C00388 V=800.0 PL=0
MOVL C00389 V=800.0 PL=0
MOVL C00390 V=800.0 PL=0
MOVL C00391 V=800.0 PL=0
MOVL C00392 V=800.0 PL=0
MOVL C00393 V=800.0 PL=0
MOVL C00394 V=800.0 PL=0
MOVL C00395 V=800.0 PL=0
MOVL C00396 V=800.0 PL=0
MOVL C00397 V=800.0 PL=0
MOVL C00398 V=800.0 PL=0
MOVL C00399 V=800.0 PL=0
MOVL C00400 V=800.0 PL=0
MOVL C00401 V=800.0 PL=0
MOVL C00402 V=800.0 PL=0
MOVL C00403 V=800.0 PL=0
MOVL C00404 V=800.0 PL=0
MOVL C00405 V=800.0 PL=0
MOVL C00406 V=800.0 PL=0
MOVL C00407 V=800.0 PL=0
MOVL C00408 V=800.0 PL=0
MOVL C00409 V=800.0 PL=0
MOVL C00410 V=800.0 PL=0
MOVL C00411 V=800.0 PL=0
MOVL C00412 V=800.0 PL=0
MOVL C00413 V=800.0 PL=0
MOVL C00414 V=800.0 PL=0
MOVL C00415 V=800.0 PL=0
MOVL C00416 V=800.0 PL=0
MOVL C00417 V=800.0 PL=0
MOVL C00418 V=800.0 PL=0
MOVL C00419 V=800.0 PL=0
MOVL C00420 V=800.0 PL=0
MOVL C00421 V=800.0 PL=0
MOVL C00422 V=800.0 PL=0
MOVL C00423 V=800.0 PL=0
MOVL C00424 V=800.0 PL=0
MOVL C00425 V=800.0 PL=0
MOVL C00426 V=800.0 PL=0
MOVL C00427 V=800.0 PL=0
MOVL C00428 V=800.0 PL=0
MOVL C00429 V=800.0 PL=0
MOVL C00430 V=800.0 PL=0
MOVL C00431 V=800.0 PL=0
MOVL C00432 V=800.0 PL=0
MOVL C00433 V=800.0 PL=0
MOVL C00434 V=800.0 PL=0
MOVL C00435 V=800.0 PL=0
MOVL C00436 V=800.0 PL=0
MOVL C00437 V=800.0 PL=0
MOVL C00438 V=800.0 PL=0
MOVL C00439 V=800.0 PL=0
MOVL C00440 V=800.0 PL=0
MOVL C00441 V=800.0 PL=0
MOVL C00442 V=800.0 PL=0
MOVL C00443 V=800.0 PL=0
MOVL C00444 V=800.0 PL=0
MOVL C00445 V=800.0 PL=0
MOVL C00446 V=800.0 PL=0
MOVL C00447 V=800.0 PL=0
MOVL C00448 V=800.0 PL=0
MOVL C00449 V=800.0 PL=0
MOVL C00450 V=800.0 PL=0
MOVL C00451 V=800.0 PL=0
MOVL C00452 V=800.0 PL=0
MOVL C00453 V=800.0 PL=0
MOVL C00454 V=800.0 PL=0
MOVL C00455 V=800.0 PL=0
MOVL C00456 V=800.0 PL=0
MOVL C00457 V=800.0 PL=0
MOVL C00458 V=800.0 PL=0
MOVL C00459 V=800.0 PL=0
MOVL C00460 V=800.0 PL=0
MOVL C00461 V=800.0 PL=0
MOVL C00462 V=800.0 PL=0
MOVL C00463 V=800.0 PL=0
MOVL C00464 V=800.0 PL=0
MOVL C00465 V=800.0 PL=0
MOVL C00466 V=800.0 PL=0
MOVL C00467 V=800.0 PL=0
MOVL C00468 V=800.0 PL=0
MOVL C00469 V=800.0 PL=0
MOVL C00470 V=800.0 PL=0
MOVL C00471 V=800.0 PL=0
MOVL C00472 V=800.0 PL=0
MOVL C00473 V=800.0 PL=0
MOVL C00474 V=800.0 PL=0
MOVL C00475 V=800.0 PL=0
MOVL C00476 V=800.0 PL=0
MOVL C00477 V=800.0 PL=0
MOVL C00478 V=800.0 PL=0
MOVL C00479 V=800.0 PL=0
MOVL C00480 V=800.0 PL=0
MOVL C00481 V=800.0 PL=0
MOVL C00482 V=800.0 PL=0
MOVL C00483 V=800.0 PL=0
MOVL C00484 V=800.0 PL=0
MOVL C00485 V=800.0 PL=0
MOVL C00486 V=800.0 PL=0
MOVL C00487 V=800.0 PL=0
MOVL C00488 V=800.0 PL=0
MOVL C00489 V=800.0 PL=0
MOVL C00490 V=800.0 PL=0
MOVL C00491 V=800.0 PL=0
MOVL C00492 V=800.0 PL=0
MOVL C00493 V=800.0 PL=0
MOVL C00494 V=800.0 PL=0
MOVL C00495 V=800.0 PL=0
MOVL C00496 V=800.0 PL=0
MOVL C00497 V=800.0 PL=0
MOVL C00498 V=800.0 PL=0
MOVL C00499 V=800.0 PL=0
MOVL C00500 V=800.0 PL=0
MOVL C00501 V=800.0 PL=0
MOVL C00502 V=800.0 PL=0
MOVL C00503 V=800.0 PL=0
MOVL C00504 V=800.0 PL=0
MOVL C00505 V=800.0 PL=0
MOVL C00506 V=800.0 PL=0
MOVL C00507 V=800.0 PL=0
MOVL C00508 V=800.0 PL=0
MOVL C00509 V=800.0 PL=0
MOVL C00510 V=800.0 PL=0
MOVL C00511 V=800.0 PL=0
MOVL C00512 V=800.0 PL=0
MOVL C00513 V=800.0 PL=0
MOVL C00514 V=800.0 PL=0
MOVL C00515 V=800.0 PL=0
MOVL C00516 V=800.0 PL=0
MOVL C00517 V=800.0 PL=0
MOVL C00518 V=800.0 PL=0
MOVL C00519 V=800.0 PL=0
MOVL C00520 V=800.0 PL=0
MOVL C00521 V=800.0 PL=0
MOVL C00522 V=800.0 PL=0
MOVL C00523 V=800.0 PL=0
MOVL C00524 V=800.0 PL=0
MOVL C00525 V=800.0 PL=0
MOVL C00526 V=800.0 PL=0
MOVL C00527 V=800.0 PL=0
MOVL C00528 V=800.0 PL=0
MOVL C00529 V=800.0 PL=0
MOVL C00530 V=800.0 PL=0
MOVL C00531 V=800.0 PL=0
MOVL C00532 V=800.0 PL=0
MOVL C00533 V=800.0 PL=0
MOVL C00534 V=800.0 PL=0
MOVL C00535 V=800.0 PL=0
MOVL C00536 V=800.0 PL=0
MOVL C00537 V=800.0 PL=0
MOVL C00538 V=800.0 PL=0
MOVL C00539 V=800.0 PL=0
MOVL C00540 V=800.0 PL=0
MOVL C00541 V=800.0 PL=0
MOVL C00542 V=800.0 PL=0
MOVL C00543 V=800.0 PL=0
MOVL C00544 V=800.0 PL=0
MOVL C00545 V=800.0 PL=0
MOVL C00546 V=800.0 PL=0
MOVL C00547 V=800.0 PL=0
MOVL C00548 V=800.0 PL=0
MOVL C00549 V=800.0 PL=0
MOVL C00550 V=800.0 PL=0
MOVL C00551 V=800.0 PL=0
MOVL C00552 V=800.0 PL=0
MOVL C00553 V=800.0 PL=0
MOVL C00554 V=800.0 PL=0
MOVL C00555 V=800.0 PL=0
MOVL C00556 V=800.0 PL=0
MOVL C00557 V=800.0 PL=0
MOVL C00558 V=800.0 PL=0
MOVL C00559 V=800.0 PL=0
MOVL C00560 V=800.0 PL=0
MOVL C00561 V=800.0 PL=0
MOVL C00562 V=800.0 PL=0
MOVL C00563 V=800.0 PL=0
MOVL C00564 V=800.0 PL=0
MOVL C00565 V=800.0 PL=0
MOVL C00566 V=800.0 PL=0
MOVL C00567 V=800.0 PL=0
MOVL C00568 V=800.0 PL=0
MOVL C00569 V=800.0 PL=0
MOVL C00570 V=800.0 PL=0
MOVL C00571 V=800.0 PL=0
MOVL C00572 V=800.0 PL=0
MOVL C00573 V=800.0 PL=0
MOVL C00574 V=800.0 PL=0
MOVL C00575 V=800.0 PL=0
MOVL C00576 V=800.0 PL=0
MOVL C00577 V=800.0 PL=0
MOVL C00578 V=800.0 PL=0
MOVL C00579 V=800.0 PL=0
MOVL C00580 V=800.0 PL=0
MOVL C00581 V=800.0 PL=0
MOVL C00582 V=800.0 PL=0
MOVL C00583 V=800.0 PL=0
MOVL C00584 V=800.0 PL=0
MOVL C00585 V=800.0 PL=0
MOVL C00586 V=800.0 PL=0
MOVL C00587 V=800.0 PL=0
MOVL C00588 V=800.0 PL=0
MOVL C00589 V=800.0 PL=0
MOVL C00590 V=800.0 PL=0
MOVL C00591 V=800.0 PL=0
MOVL C00592 V=800.0 PL=0
MOVL C00593 V=800.0 PL=0
MOVL C00594 V=800.0 PL=0
MOVL C00595 V=800.0 PL=0
MOVL C00596 V=800.0 PL=0
MOVL C00597 V=800.0 PL=0
MOVL C00598 V=800.0 PL=0
MOVL C00599 V=800.0 PL=0
MOVL C00600 V=800.0 PL=0
MOVL C00601 V=800.0 PL=0
MOVL C00602 V=800.0 PL=0
MOVL C00603 V=800.0 PL=0
MOVL C00604 V=800.0 PL=0
MOVL C00605 V=800.0 PL=0
MOVL C00606 V=800.0 PL=0
MOVL C00607 V=800.0 PL=0
MOVL C00608 V=800.0 PL=0
MOVL C00609 V=800.0 PL=0
MOVL C00610 V=800.0 PL=0
MOVL C00611 V=800.0 PL=0
MOVL C00612 V=800.0 PL=0
MOVL C00613 V=800.0 PL=0
MOVL C00614 V=800.0 PL=0
MOVL C00615 V=800.0 PL=0
MOVL C00616 V=800.0 PL=0
MOVL C00617 V=800.0 PL=0
MOVL C00618 V=800.0 PL=0
MOVL C00619 V=800.0 PL=0
MOVL C00620 V=800.0 PL=0
MOVL C00621 V=800.0 PL=0
MOVL C00622 V=800.0 PL=0
MOVL C00623 V=800.0 PL=0
MOVL C00624 V=800.0 PL=0
MOVL C00625 V=800.0 PL=0
MOVL C00626 V=800.0 PL=0
MOVL C00627 V=800.0 PL=0
MOVL C00628 V=800.0 PL=0
MOVL C00629 V=800.0 PL=0
MOVL C00630 V=800.0 PL=0
MOVL C00631 V=800.0 PL=0
MOVL C00632 V=800.0 PL=0
MOVL C00633 V=800.0 PL=0
MOVL C00634 V=800.0 PL=0
MOVL C00635 V=800.0 PL=0
MOVL C00636 V=800.0 PL=0
MOVL C00637 V=800.0 PL=0
MOVL C00638 V=800.0 PL=0
MOVL C00639 V=800.0 PL=0
MOVL C00640 V=800.0 PL=0
MOVL C00641 V=800.0 PL=0
MOVL C00642 V=800.0 PL=0
MOVL C00643 V=800.0 PL=0
MOVL C00644 V=800.0 PL=0
MOVL C00645 V=800.0 PL=0
MOVL C00646 V=800.0 PL=0
MOVL C00647 V=800.0 PL=0
MOVL C00648 V=800.0 PL=0
MOVL C00649 V=800.0 PL=0
MOVL C00650 V=800.0 PL=0
MOVL C00651 V=800.0 PL=0
MOVL C00652 V=800.0 PL=0
MOVL C00653 V=800.0 PL=0
MOVL C00654 V=800.0 PL=0
MOVL C00655 V=800.0 PL=0
MOVL C00656 V=800.0 PL=0
MOVL C00657 V=800.0 PL=0
MOVL C00658 V=800.0 PL=0
MOVL C00659 V=800.0 PL=0
MOVL C00660 V=800.0 PL=0
MOVL C00661 V=800.0 PL=0
MOVL C00662 V=800.0 PL=0
MOVL C00663 V=800.0 PL=0
MOVL C00664 V=800.0 PL=0
MOVL C00665 V=800.0 PL=0
MOVL C00666 V=800.0 PL=0
MOVL C00667 V=800.0 PL=0
MOVL C00668 V=800.0 PL=0
MOVL C00669 V=800.0 PL=0
MOVL C00670 V=800.0 PL=0
MOVL C00671 V=800.0 PL=0
MOVL C00672 V=800.0 PL=0
MOVL C00673 V=800.0 PL=0
MOVL C00674 V=800.0 PL=0
MOVL C00675 V=800.0 PL=0
MOVL C00676 V=800.0 PL=0
MOVL C00677 V=800.0 PL=0
MOVL C00678 V=800.0 PL=0
MOVL C00679 V=800.0 PL=0
MOVL C00680 V=800.0 PL=0
MOVL C00681 V=800.0 PL=0
MOVL C00682 V=800.0 PL=0
MOVL C00683 V=800.0 PL=0
MOVL C00684 V=800.0 PL=0
MOVL C00685 V=800.0 PL=0
MOVL C00686 V=800.0 PL=0
MOVL C00687 V=800.0 PL=0
MOVL C00688 V=800.0 PL=0
MOVL C00689 V=800.0 PL=0
MOVL C00690 V=800.0 PL=0
MOVL C00691 V=800.0 PL=0
MOVL C00692 V=800.0 PL=0
MOVL C00693 V=800.0 PL=0
MOVL C00694 V=800.0 PL=0
MOVL C00695 V=800.0 PL=0
MOVL C00696 V=800.0 PL=0
MOVL C00697 V=800.0 PL=0
MOVL C00698 V=800.0 PL=0
MOVL C00699 V=800.0 PL=0
MOVL C00700 V=800.0 PL=0
MOVL C00701 V=800.0 PL=0
MOVL C00702 V=800.0 PL=0
MOVL C00703 V=800.0 PL=0
MOVL C00704 V=800.0 PL=0
MOVL C00705 V=800.0 PL=0
MOVL C00706 V=800.0 PL=0
MOVL C00707 V=800.0 PL=0
MOVL C00708 V=800.0 PL=0
MOVL C00709 V=800.0 PL=0
MOVL C00710 V=800.0 PL=0
MOVL C00711 V=800.0 PL=0
MOVL C00712 V=800.0 PL=0
MOVL C00713 V=800.0 PL=0
MOVL C00714 V=800.0 PL=0
MOVL C00715 V=800.0 PL=0
MOVL C00716 V=800.0 PL=0
MOVL C00717 V=800.0 PL=0
MOVL C00718 V=800.0 PL=0
MOVL C00719 V=800.0 PL=0
MOVL C00720 V=800.0 PL=0
MOVL C00721 V=800.0 PL=0
MOVL C00722 V=800.0 PL=0
MOVL C00723 V=800.0 PL=0
MOVL C00724 V=800.0 PL=0
MOVL C00725 V=800.0 PL=0
MOVL C00726 V=800.0 PL=0
MOVL C00727 V=800.0 PL=0
MOVL C00728 V=800.0 PL=0
MOVL C00729 V=800.0 PL=0
MOVL C00730 V=800.0 PL=0
MOVL C00731 V=800.0 PL=0
MOVL C00732 V=800.0 PL=0
MOVL C00733 V=800.0 PL=0
MOVL C00734 V=800.0 PL=0
MOVL C00735 V=800.0 PL=0
MOVL C00736 V=800.0 PL=0
MOVL C00737 V=800.0 PL=0
MOVL C00738 V=800.0 PL=0
MOVL C00739 V=800.0 PL=0
MOVL C00740 V=800.0 PL=0
MOVL C00741 V=800.0 PL=0
MOVL C00742 V=800.0 PL=0
MOVL C00743 V=800.0 PL=0
MOVL C00744 V=800.0 PL=0
MOVL C00745 V=800.0 PL=0
MOVL C00746 V=800.0 PL=0
MOVL C00747 V=800.0 PL=0
MOVL C00748 V=800.0 PL=0
MOVL C00749 V=800.0 PL=0
MOVL C00750 V=800.0 PL=0
MOVL C00751 V=800.0 PL=0
MOVL C00752 V=800.0 PL=0
MOVL C00753 V=800.0 PL=0
MOVL C00754 V=800.0 PL=0
MOVL C00755 V=800.0 PL=0
MOVL C00756 V=800.0 PL=0
MOVL C00757 V=800.0 PL=0
MOVL C00758 V=800.0 PL=0
MOVL C00759 V=800.0 PL=0
MOVL C00760 V=800.0 PL=0
MOVL C00761 V=800.0 PL=0
MOVL C00762 V=800.0 PL=0
MOVL C00763 V=800.0 PL=0
MOVL C00764 V=800.0 PL=0
MOVL C00765 V=800.0 PL=0
MOVL C00766 V=800.0 PL=0
MOVL C00767 V=800.0 PL=0
MOVL C00768 V=800.0 PL=0
MOVL C00769 V=800.0 PL=0
MOVL C00770 V=800.0 PL=0
MOVL C00771 V=800.0 PL=0
MOVL C00772 V=800.0 PL=0
MOVL C00773 V=800.0 PL=0
MOVL C00774 V=800.0 PL=0
MOVL C00775 V=800.0 PL=0
MOVL C00776 V=800.0 PL=0
MOVL C00777 V=800.0 PL=0
MOVL C00778 V=800.0 PL=0
MOVL C00779 V=800.0 PL=0
MOVL C00780 V=800.0 PL=0
MOVL C00781 V=800.0 PL=0
MOVL C00782 V=800.0 PL=0
MOVL C00783 V=800.0 PL=0
MOVL C00784 V=800.0 PL=0
MOVL C00785 V=800.0 PL=0
MOVL C00786 V=800.0 PL=0
MOVL C00787 V=800.0 PL=0
MOVL C00788 V=800.0 PL=0
MOVL C00789 V=800.0 PL=0
MOVL C00790 V=800.0 PL=0
MOVL C00791 V=800.0 PL=0
MOVL C00792 V=800.0 PL=0
MOVL C00793 V=800.0 PL=0
MOVL C00794 V=800.0 PL=0
MOVL C00795 V=800.0 PL=0
MOVL C00796 V=800.0 PL=0
MOVL C00797 V=800.0 PL=0
MOVL C00798 V=800.0 PL=0
MOVL C00799 V=800.0 PL=0
MOVL C00800 V=800.0 PL=0
MOVL C00801 V=800.0 PL=0
MOVL C00802 V=800.0 PL=0
MOVL C00803 V=800.0 PL=0
MOVL C00804 V=800.0 PL=0
MOVL C00805 V=800.0 PL=0
MOVL C00806 V=800.0 PL=0
MOVL C00807 V=800.0 PL=0
MOVL C00808 V=800.0 PL=0
MOVL C00809 V=800.0 PL=0
MOVL C00810 V=800.0 PL=0
MOVL C00811 V=800.0 PL=0
MOVL C00812 V=800.0 PL=0
MOVL C00813 V=800.0 PL=0
MOVL C00814 V=800.0 PL=0
MOVL C00815 V=800.0 PL=0
MOVL C00816 V=800.0 PL=0
MOVL C00817 V=800.0 PL=0
MOVL C00818 V=800.0 PL=0
MOVL C00819 V=800.0 PL=0
MOVL C00820 V=800.0 PL=0
MOVL C00821 V=800.0 PL=0
MOVL C00822 V=800.0 PL=0
MOVL C00823 V=800.0 PL=0
MOVL C00824 V=800.0 PL=0
MOVL C00825 V=800.0 PL=0
MOVL C00826 V=800.0 PL=0
MOVL C00827 V=800.0 PL=0
MOVL C00828 V=800.0 PL=0
MOVL C00829 V=800.0 PL=0
MOVL C00830 V=800.0 PL=0
MOVL C00831 V=800.0 PL=0
MOVL C00832 V=800.0 PL=0
MOVL C00833 V=800.0 PL=0
MOVL C00834 V=800.0 PL=0
MOVL C00835 V=800.0 PL=0
MOVL C00836 V=800.0 PL=0
MOVL C00837 V=800.0 PL=0
MOVL C00838 V=800.0 PL=0
MOVL C00839 V=800.0 PL=0
MOVL C00840 V=800.0 PL=0
MOVL C00841 V=800.0 PL=0
MOVL C00842 V=800.0 PL=0
MOVL C00843 V=800.0 PL=0
MOVL C00844 V=800.0 PL=0
MOVL C00845 V=800.0 PL=0
MOVL C00846 V=800.0 PL=0
MOVL C00847 V=800.0 PL=0
MOVL C00848 V=800.0 PL=0
MOVL C00849 V=800.0 PL=0
MOVL C00850 V=800.0 PL=0
MOVL C00851 V=800.0 PL=0
MOVL C00852 V=800.0 PL=0
MOVL C00853 V=800.0 PL=0
MOVL C00854 V=800.0 PL=0
MOVL C00855 V=800.0 PL=0
MOVL C00856 V=800.0 PL=0
MOVL C00857 V=800.0 PL=0
MOVL C00858 V=800.0 PL=0
MOVL C00859 V=800.0 PL=0
MOVL C00860 V=800.0 PL=0
MOVL C00861 V=800.0 PL=0
MOVL C00862 V=800.0 PL=0
MOVL C00863 V=800.0 PL=0
MOVL C00864 V=800.0 PL=0
MOVL C00865 V=800.0 PL=0
MOVL C00866 V=800.0 PL=0
MOVL C00867 V=800.0 PL=0
MOVL C00868 V=800.0 PL=0
MOVL C00869 V=800.0 PL=0
MOVL C00870 V=800.0 PL=0
MOVL C00871 V=800.0 PL=0
MOVL C00872 V=800.0 PL=0
MOVL C00873 V=800.0 PL=0
MOVL C00874 V=800.0 PL=0
MOVL C00875 V=800.0 PL=0
MOVL C00876 V=800.0 PL=0
MOVL C00877 V=800.0 PL=0
MOVL C00878 V=800.0 PL=0
MOVL C00879 V=800.0 PL=0
MOVL C00880 V=800.0 PL=0
MOVL C00881 V=800.0 PL=0
MOVL C00882 V=800.0 PL=0
MOVL C00883 V=800.0 PL=0
MOVL C00884 V=800.0 PL=0
MOVL C00885 V=800.0 PL=0
MOVL C00886 V=800.0 PL=0
MOVL C00887 V=800.0 PL=0
MOVL C00888 V=800.0 PL=0
MOVL C00889 V=800.0 PL=0
MOVL C00890 V=800.0 PL=0
MOVL C00891 V=800.0 PL=0
MOVL C00892 V=800.0 PL=0
MOVL C00893 V=800.0 PL=0
MOVL C00894 V=800.0 PL=0
MOVL C00895 V=800.0 PL=0
MOVL C00896 V=800.0 PL=0
MOVL C00897 V=800.0 PL=0
MOVL C00898 V=800.0 PL=0
MOVL C00899 V=800.0 PL=0
MOVL C00900 V=800.0 PL=0
MOVL C00901 V=800.0 PL=0
MOVL C00902 V=800.0 PL=0
MOVL C00903 V=800.0 PL=0
MOVL C00904 V=800.0 PL=0
MOVL C00905 V=800.0 PL=0
MOVL C00906 V=800.0 PL=0
MOVL C00907 V=800.0 PL=0
MOVL C00908 V=800.0 PL=0
MOVL C00909 V=800.0 PL=0
MOVL C00910 V=800.0 PL=0
MOVL C00911 V=800.0 PL=0
MOVL C00912 V=800.0 PL=0
MOVL C00913 V=800.0 PL=0
MOVL C00914 V=800.0 PL=0
MOVL C00915 V=800.0 PL=0
MOVL C00916 V=800.0 PL=0
MOVL C00917 V=800.0 PL=0
MOVL C00918 V=800.0 PL=0
MOVL C00919 V=800.0 PL=0
MOVL C00920 V=800.0 PL=0
MOVL C00921 V=800.0 PL=0
MOVL C00922 V=800.0 PL=0
MOVL C00923 V=800.0 PL=0
MOVL C00924 V=800.0 PL=0
MOVL C00925 V=800.0 PL=0
MOVL C00926 V=800.0 PL=0
MOVL C00927 V=800.0 PL=0
MOVL C00928 V=800.0 PL=0
MOVL C00929 V=800.0 PL=0
MOVL C00930 V=800.0 PL=0
MOVL C00931 V=800.0 PL=0
MOVL C00932 V=800.0 PL=0
MOVL C00933 V=800.0 PL=0
MOVL C00934 V=800.0 PL=0
MOVL C00935 V=800.0 PL=0
MOVL C00936 V=800.0 PL=0
MOVL C00937 V=800.0 PL=0
MOVL C00938 V=800.0 PL=0
MOVL C00939 V=800.0 PL=0
MOVL C00940 V=800.0 PL=0
MOVL C00941 V=800.0 PL=0
MOVL C00942 V=800.0 PL=0
MOVL C00943 V=800.0 PL=0
MOVL C00944 V=800.0 PL=0
MOVL C00945 V=800.0 PL=0
MOVL C00946 V=800.0 PL=0
MOVL C00947 V=800.0 PL=0
MOVL C00948 V=800.0 PL=0
MOVL C00949 V=800.0 PL=0
MOVL C00950 V=800.0 PL=0
MOVL C00951 V=800.0 PL=0
MOVL C00952 V=800.0 PL=0
MOVL C00953 V=800.0 PL=0
MOVL C00954 V=800.0 PL=0
MOVL C00955 V=800.0 PL=0
MOVL C00956 V=800.0 PL=0
MOVL C00957 V=800.0 PL=0
MOVL C00958 V=800.0 PL=0
MOVL C00959 V=800.0 PL=0
MOVL C00960 V=800.0 PL=0
MOVL C00961 V=800.0 PL=0
MOVL C00962 V=800.0 PL=0
MOVL C00963 V=800.0 PL=0
MOVL C00964 V=800.0 PL=0
MOVL C00965 V=800.0 PL=0
MOVL C00966 V=800.0 PL=0
MOVL C00967 V=800.0 PL=0
MOVL C00968 V=800.0 PL=0
MOVL C00969 V=800.0 PL=0
MOVL C00970 V=800.0 PL=0
MOVL C00971 V=800.0 PL=0
MOVL C00972 V=800.0 PL=0
MOVL C00973 V=800.0 PL=0
MOVL C00974 V=800.0 PL=0
MOVL C00975 V=800.0 PL=0
MOVL C00976 V=800.0 PL=0
MOVL C00977 V=800.0 PL=0
MOVL C00978 V=800.0 PL=0
MOVL C00979 V=800.0 PL=0
MOVL C00980 V=800.0 PL=0
MOVL C00981 V=800.0 PL=0
MOVL C00982 V=800.0 PL=0
MOVL C00983 V=800.0 PL=0
MOVL C00984 V=800.0 PL=0
MOVL C00985 V=800.0 PL=0
MOVL C00986 V=800.0 PL=0
MOVL C00987 V=800.0 PL=0
MOVL C00988 V=800.0 PL=0
MOVL C00989 V=800.0 PL=0
MOVL C00990 V=800.0 PL=0
MOVL C00991 V=800.0 PL=0
MOVL C00992 V=800.0 PL=0
MOVL C00993 V=800.0 PL=0
MOVL C00994 V=800.0 PL=0
MOVL C00995 V=800.0 PL=0
MOVL C00996 V=800.0 PL=0
MOVL C00997 V=800.0 PL=0
MOVL C00998 V=800.0 PL=0
MOVL C00999 V=800.0 PL=0
MOVL C01000 V=800.0 PL=0
MOVL C01001 V=800.0 PL=0
MOVL C01002 V=800.0 PL=0
MOVL C01003 V=800.0 PL=0
MOVL C01004 V=800.0 PL=0
MOVL C01005 V=800.0 PL=0
MOVL C01006 V=800.0 PL=0
MOVL C01007 V=800.0 PL=0
MOVL C01008 V=800.0 PL=0
MOVL C01009 V=800.0 PL=0
MOVL C01010 V=800.0 PL=0
MOVL C01011 V=800.0 PL=0
MOVL C01012 V=800.0 PL=0
MOVL C01013 V=800.0 PL=0
MOVL C01014 V=800.0 PL=0
MOVL C01015 V=800.0 PL=0
MOVL C01016 V=800.0 PL=0
MOVL C01017 V=800.0 PL=0
MOVL C01018 V=800.0 PL=0
MOVL C01019 V=800.0 PL=0
MOVL C01020 V=800.0 PL=0
MOVL C01021 V=800.0 PL=0
MOVL C01022 V=800.0 PL=0
MOVL C01023 V=800.0 PL=0
MOVL C01024 V=800.0 PL=0
MOVL C01025 V=800.0 PL=0
MOVL C01026 V=800.0 PL=0
MOVL C01027 V=800.0 PL=0
MOVL C01028 V=800.0 PL=0
MOVL C01029 V=800.0 PL=0
MOVL C01030 V=800.0 PL=0
MOVL C01031 V=800.0 PL=0
MOVL C01032 V=800.0 PL=0
MOVL C01033 V=800.0 PL=0
MOVL C01034 V=800.0 PL=0
MOVL C01035 V=800.0 PL=0
MOVL C01036 V=800.0 PL=0
MOVL C01037 V=800.0 PL=0
MOVL C01038 V=800.0 PL=0
MOVL C01039 V=800.0 PL=0
MOVL C01040 V=800.0 PL=0
MOVL C01041 V=800.0 PL=0
MOVL C01042 V=800.0 PL=0
MOVL C01043 V=800.0 PL=0
MOVL C01044 V=800.0 PL=0
MOVL C01045 V=800.0 PL=0
MOVL C01046 V=800.0 PL=0
MOVL C01047 V=800.0 PL=0
MOVL C01048 V=800.0 PL=0
MOVL C01049 V=800.0 PL=0
MOVL C01050 V=800.0 PL=0
MOVL C01051 V=800.0 PL=0
MOVL C01052 V=800.0 PL=0
MOVL C01053 V=800.0 PL=0
MOVL C01054 V=800.0 PL=0
MOVL C01055 V=800.0 PL=0
MOVL C01056 V=800.0 PL=0
MOVL C01057 V=800.0 PL=0
MOVL C01058 V=800.0 PL=0
MOVL C01059 V=800.0 PL=0
MOVL C01060 V=800.0 PL=0
MOVL C01061 V=800.0 PL=0
MOVL C01062 V=800.0 PL=0
MOVL C01063 V=800.0 PL=0
MOVL C01064 V=800.0 PL=0
MOVL C01065 V=800.0 PL=0
MOVL C01066 V=800.0 PL=0
MOVL C01067 V=800.0 PL=0
MOVL C01068 V=800.0 PL=0
MOVL C01069 V=800.0 PL=0
MOVL C01070 V=800.0 PL=0
MOVL C01071 V=800.0 PL=0
MOVL C01072 V=800.0 PL=0
MOVL C01073 V=800.0 PL=0
MOVL C01074 V=800.0 PL=0
MOVL C01075 V=800.0 PL=0
MOVL C01076 V=800.0 PL=0
MOVL C01077 V=800.0 PL=0
MOVL C01078 V=800.0 PL=0
MOVL C01079 V=800.0 PL=0
MOVL C01080 V=800.0 PL=0
MOVL C01081 V=800.0 PL=0
MOVL C01082 V=800.0 PL=0
MOVL C01083 V=800.0 PL=0
MOVL C01084 V=800.0 PL=0
MOVL C01085 V=800.0 PL=0
MOVL C01086 V=800.0 PL=0
MOVL C01087 V=800.0 PL=0
MOVL C01088 V=800.0 PL=0
MOVL C01089 V=800.0 PL=0
MOVL C01090 V=800.0 PL=0
MOVL C01091 V=800.0 PL=0
MOVL C01092 V=800.0 PL=0
MOVL C01093 V=800.0 PL=0
MOVL C01094 V=800.0 PL=0
MOVL C01095 V=800.0 PL=0
MOVL C01096 V=800.0 PL=0
MOVL C01097 V=800.0 PL=0
MOVL C01098 V=800.0 PL=0
MOVL C01099 V=800.0 PL=0
MOVL C01100 V=800.0 PL=0
MOVL C01101 V=800.0 PL=0
MOVL C01102 V=800.0 PL=0
MOVL C01103 V=800.0 PL=0
MOVL C01104 V=800.0 PL=0
MOVL C01105 V=800.0 PL=0
MOVL C01106 V=800.0 PL=0
MOVL C01107 V=800.0 PL=0
MOVL C01108 V=800.0 PL=0
MOVL C01109 V=800.0 PL=0
MOVL C01110 V=800.0 PL=0
MOVL C01111 V=800.0 PL=0
MOVL C01112 V=800.0 PL=0
MOVL C01113 V=800.0 PL=0
MOVL C01114 V=800.0 PL=0
MOVL C01115 V=800.0 PL=0
MOVL C01116 V=800.0 PL=0
MOVL C01117 V=800.0 PL=0
MOVL C01118 V=800.0 PL=0
MOVL C01119 V=800.0 PL=0
MOVL C01120 V=800.0 PL=0
MOVL C01121 V=800.0 PL=0
MOVL C01122 V=800.0 PL=0
MOVL C01123 V=800.0 PL=0
MOVL C01124 V=800.0 PL=0
MOVL C01125 V=800.0 PL=0
MOVL C01126 V=800.0 PL=0
MOVL C01127 V=800.0 PL=0
MOVL C01128 V=800.0 PL=0
MOVL C01129 V=800.0 PL=0
MOVL C01130 V=800.0 PL=0
MOVL C01131 V=800.0 PL=0
MOVL C01132 V=800.0 PL=0
MOVL C01133 V=800.0 PL=0
MOVL C01134 V=800.0 PL=0
MOVL C01135 V=800.0 PL=0
MOVL C01136 V=800.0 PL=0
MOVL C01137 V=800.0 PL=0
MOVL C01138 V=800.0 PL=0
MOVL C01139 V=800.0 PL=0
MOVL C01140 V=800.0 PL=0
MOVL C01141 V=800.0 PL=0
MOVL C01142 V=800.0 PL=0
MOVL C01143 V=800.0 PL=0
MOVL C01144 V=800.0 PL=0
MOVL C01145 V=800.0 PL=0
MOVL C01146 V=800.0 PL=0
MOVL C01147 V=800.0 PL=0
MOVL C01148 V=800.0 PL=0
MOVL C01149 V=800.0 PL=0
MOVL C01150 V=800.0 PL=0
MOVL C01151 V=800.0 PL=0
MOVL C01152 V=800.0 PL=0
MOVL C01153 V=800.0 PL=0
MOVL C01154 V=800.0 PL=0
MOVL C01155 V=800.0 PL=0
MOVL C01156 V=800.0 PL=0
MOVL C01157 V=800.0 PL=0
MOVL C01158 V=800.0 PL=0
MOVL C01159 V=800.0 PL=0
MOVL C01160 V=800.0 PL=0
MOVL C01161 V=800.0 PL=0
MOVL C01162 V=800.0 PL=0
MOVL C01163 V=800.0 PL=0
MOVL C01164 V=800.0 PL=0
MOVL C01165 V=800.0 PL=0
MOVL C01166 V=800.0 PL=0
MOVL C01167 V=800.0 PL=0
MOVL C01168 V=800.0 PL=0
MOVL C01169 V=800.0 PL=0
MOVL C01170 V=800.0 PL=0
MOVL C01171 V=800.0 PL=0
MOVL C01172 V=800.0 PL=0
MOVL C01173 V=800.0 PL=0
MOVL C01174 V=800.0 PL=0
MOVL C01175 V=800.0 PL=0
MOVL C01176 V=800.0 PL=0
MOVL C01177 V=800.0 PL=0
MOVL C01178 V=800.0 PL=0
MOVL C01179 V=800.0 PL=0
MOVL C01180 V=800.0 PL=0
MOVL C01181 V=800.0 PL=0
MOVL C01182 V=800.0 PL=0
MOVL C01183 V=800.0 PL=0
MOVL C01184 V=800.0 PL=0
MOVL C01185 V=800.0 PL=0
MOVL C01186 V=800.0 PL=0
MOVL C01187 V=800.0 PL=0
MOVL C01188 V=800.0 PL=0
MOVL C01189 V=800.0 PL=0
MOVL C01190 V=800.0 PL=0
MOVL C01191 V=800.0 PL=0
MOVL C01192 V=800.0 PL=0
MOVL C01193 V=800.0 PL=0
MOVL C01194 V=800.0 PL=0
MOVL C01195 V=800.0 PL=0
MOVL C01196 V=800.0 PL=0
MOVL C01197 V=800.0 PL=0
MOVL C01198 V=800.0 PL=0
MOVL C01199 V=800.0 PL=0
MOVL C01200 V=800.0 PL=0
MOVL C01201 V=800.0 PL=0
MOVL C01202 V=800.0 PL=0
MOVL C01203 V=800.0 PL=0
MOVL C01204 V=800.0 PL=0
MOVL C01205 V=800.0 PL=0
MOVL C01206 V=800.0 PL=0
MOVL C01207 V=800.0 PL=0
MOVL C01208 V=800.0 PL=0
MOVL C01209 V=800.0 PL=0
MOVL C01210 V=800.0 PL=0
MOVL C01211 V=800.0 PL=0
MOVL C01212 V=800.0 PL=0
MOVL C01213 V=800.0 PL=0
MOVL C01214 V=800.0 PL=0
MOVL C01215 V=800.0 PL=0
MOVL C01216 V=800.0 PL=0
MOVL C01217 V=800.0 PL=0
MOVL C01218 V=800.0 PL=0
MOVL C01219 V=800.0 PL=0
MOVL C01220 V=800.0 PL=0
MOVL C01221 V=800.0 PL=0
MOVL C01222 V=800.0 PL=0
MOVL C01223 V=800.0 PL=0
MOVL C01224 V=800.0 PL=0
MOVL C01225 V=800.0 PL=0
MOVL C01226 V=800.0 PL=0
MOVL C01227 V=800.0 PL=0
MOVL C01228 V=800.0 PL=0
MOVL C01229 V=800.0 PL=0
MOVL C01230 V=800.0 PL=0
MOVL C01231 V=800.0 PL=0
MOVL C01232 V=800.0 PL=0
MOVL C01233 V=800.0 PL=0
MOVL C01234 V=800.0 PL=0
MOVL C01235 V=800.0 PL=0
MOVL C01236 V=800.0 PL=0
MOVL C01237 V=800.0 PL=0
MOVL C01238 V=800.0 PL=0
MOVL C01239 V=800.0 PL=0
MOVL C01240 V=800.0 PL=0
MOVL C01241 V=800.0 PL=0
MOVL C01242 V=800.0 PL=0
MOVL C01243 V=800.0 PL=0
MOVL C01244 V=800.0 PL=0
MOVL C01245 V=800.0 PL=0
MOVL C01246 V=800.0 PL=0
MOVL C01247 V=800.0 PL=0
MOVL C01248 V=800.0 PL=0
MOVL C01249 V=800.0 PL=0
MOVL C01250 V=800.0 PL=0
MOVL C01251 V=800.0 PL=0
MOVL C01252 V=800.0 PL=0
MOVL C01253 V=800.0 PL=0
MOVL C01254 V=800.0 PL=0
MOVL C01255 V=800.0 PL=0
MOVL C01256 V=800.0 PL=0
MOVL C01257 V=800.0 PL=0
MOVL C01258 V=800.0 PL=0
MOVL C01259 V=800.0 PL=0
MOVL C01260 V=800.0 PL=0
MOVL C01261 V=800.0 PL=0
MOVL C01262 V=800.0 PL=0
MOVL C01263 V=800.0 PL=0
MOVL C01264 V=800.0 PL=0
MOVL C01265 V=800.0 PL=0
MOVL C01266 V=800.0 PL=0
MOVL C01267 V=800.0 PL=0
MOVL C01268 V=800.0 PL=0
MOVL C01269 V=800.0 PL=0
MOVL C01270 V=800.0 PL=0
MOVL C01271 V=800.0 PL=0
MOVL C01272 V=800.0 PL=0
MOVL C01273 V=800.0 PL=0
MOVL C01274 V=800.0 PL=0
MOVL C01275 V=800.0 PL=0
MOVL C01276 V=800.0 PL=0
MOVL C01277 V=800.0 PL=0
MOVL C01278 V=800.0 PL=0
MOVL C01279 V=800.0 PL=0
MOVL C01280 V=800.0 PL=0
MOVL C01281 V=800.0 PL=0
MOVL C01282 V=800.0 PL=0
MOVL C01283 V=800.0 PL=0
MOVL C01284 V=800.0 PL=0
MOVL C01285 V=800.0 PL=0
MOVL C01286 V=800.0 PL=0
MOVL C01287 V=800.0 PL=0
MOVL C01288 V=800.0 PL=0
MOVL C01289 V=800.0 PL=0
MOVL C01290 V=800.0 PL=0
MOVL C01291 V=800.0 PL=0
MOVL C01292 V=800.0 PL=0
MOVL C01293 V=800.0 PL=0
MOVL C01294 V=800.0 PL=0
MOVL C01295 V=800.0 PL=0
MOVL C01296 V=800.0 PL=0
MOVL C01297 V=800.0 PL=0
MOVL C01298 V=800.0 PL=0
MOVL C01299 V=800.0 PL=0
MOVL C01300 V=800.0 PL=0
MOVL C01301 V=800.0 PL=0
MOVL C01302 V=800.0 PL=0
MOVL C01303 V=800.0 PL=0
MOVL C01304 V=800.0 PL=0
MOVL C01305 V=800.0 PL=0
MOVL C01306 V=800.0 PL=0
MOVL C01307 V=800.0 PL=0
MOVL C01308 V=800.0 PL=0
MOVL C01309 V=800.0 PL=0
MOVL C01310 V=800.0 PL=0
MOVL C01311 V=800.0 PL=0
MOVL C01312 V=800.0 PL=0
MOVL C01313 V=800.0 PL=0
MOVL C01314 V=800.0 PL=0
MOVL C01315 V=800.0 PL=0
MOVL C01316 V=800.0 PL=0
MOVL C01317 V=800.0 PL=0
MOVL C01318 V=800.0 PL=0
MOVL C01319 V=800.0 PL=0
MOVL C01320 V=800.0 PL=0
MOVL C01321 V=800.0 PL=0
MOVL C01322 V=800.0 PL=0
MOVL C01323 V=800.0 PL=0
MOVL C01324 V=800.0 PL=0
MOVL C01325 V=800.0 PL=0
MOVL C01326 V=800.0 PL=0
MOVL C01327 V=800.0 PL=0
MOVL C01328 V=800.0 PL=0
MOVL C01329 V=800.0 PL=0
MOVL C01330 V=800.0 PL=0
MOVL C01331 V=800.0 PL=0
MOVL C01332 V=800.0 PL=0
MOVL C01333 V=800.0 PL=0
MOVL C01334 V=800.0 PL=0
MOVL C01335 V=800.0 PL=0
MOVL C01336 V=800.0 PL=0
MOVL C01337 V=800.0 PL=0
MOVL C01338 V=800.0 PL=0
MOVL C01339 V=800.0 PL=0
MOVL C01340 V=800.0 PL=0
MOVL C01341 V=800.0 PL=0
MOVL C01342 V=800.0 PL=0
MOVL C01343 V=800.0 PL=0
MOVL C01344 V=800.0 PL=0
MOVL C01345 V=800.0 PL=0
MOVL C01346 V=800.0 PL=0
MOVL C01347 V=800.0 PL=0
MOVL C01348 V=800.0 PL=0
MOVL C01349 V=800.0 PL=0
MOVL C01350 V=800.0 PL=0
MOVL C01351 V=800.0 PL=0
MOVL C01352 V=800.0 PL=0
MOVL C01353 V=800.0 PL=0
MOVL C01354 V=800.0 PL=0
MOVL C01355 V=800.0 PL=0
MOVL C01356 V=800.0 PL=0
MOVL C01357 V=800.0 PL=0
MOVL C01358 V=800.0 PL=0
MOVL C01359 V=800.0 PL=0
MOVL C01360 V=800.0 PL=0
MOVL C01361 V=800.0 PL=0
MOVL C01362 V=800.0 PL=0
MOVL C01363 V=800.0 PL=0
MOVL C01364 V=800.0 PL=0
MOVL C01365 V=800.0 PL=0
MOVL C01366 V=800.0 PL=0
MOVL C01367 V=800.0 PL=0
MOVL C01368 V=800.0 PL=0
MOVL C01369 V=800.0 PL=0
MOVL C01370 V=800.0 PL=0
MOVL C01371 V=800.0 PL=0
MOVL C01372 V=800.0 PL=0
MOVL C01373 V=800.0 PL=0
MOVL C01374 V=800.0 PL=0
MOVL C01375 V=800.0 PL=0
MOVL C01376 V=800.0 PL=0
MOVL C01377 V=800.0 PL=0
MOVL C01378 V=800.0 PL=0
MOVL C01379 V=800.0 PL=0
MOVL C01380 V=800.0 PL=0
MOVL C01381 V=800.0 PL=0
MOVL C01382 V=800.0 PL=0
MOVL C01383 V=800.0 PL=0
MOVL C01384 V=800.0 PL=0
MOVL C01385 V=800.0 PL=0
MOVL C01386 V=800.0 PL=0
MOVL C01387 V=800.0 PL=0
MOVL C01388 V=800.0 PL=0
MOVL C01389 V=800.0 PL=0
MOVL C01390 V=800.0 PL=0
MOVL C01391 V=800.0 PL=0
MOVL C01392 V=800.0 PL=0
MOVL C01393 V=800.0 PL=0
MOVL C01394 V=800.0 PL=0
MOVL C01395 V=800.0 PL=0
MOVL C01396 V=800.0 PL=0
MOVL C01397 V=800.0 PL=0
MOVL C01398 V=800.0 PL=0
MOVL C01399 V=800.0 PL=0
MOVL C01400 V=800.0 PL=0
MOVL C01401 V=800.0 PL=0
MOVL C01402 V=800.0 PL=0
MOVL C01403 V=800.0 PL=0
MOVL C01404 V=800.0 PL=0
MOVL C01405 V=800.0 PL=0
MOVL C01406 V=800.0 PL=0
MOVL C01407 V=800.0 PL=0
MOVL C01408 V=800.0 PL=0
MOVL C01409 V=800.0 PL=0
MOVL C01410 V=800.0 PL=0
MOVL C01411 V=800.0 PL=0
MOVL C01412 V=800.0 PL=0
MOVL C01413 V=800.0 PL=0
MOVL C01414 V=800.0 PL=0
MOVL C01415 V=800.0 PL=0
MOVL C01416 V=800.0 PL=0
MOVL C01417 V=800.0 PL=0
MOVL C01418 V=800.0 PL=0
MOVL C01419 V=800.0 PL=0
MOVL C01420 V=800.0 PL=0
MOVL C01421 V=800.0 PL=0
MOVL C01422 V=800.0 PL=0
MOVL C01423 V=800.0 PL=0
MOVL C01424 V=800.0 PL=0
MOVL C01425 V=800.0 PL=0
MOVL C01426 V=800.0 PL=0
MOVL C01427 V=800.0 PL=0
MOVL C01428 V=800.0 PL=0
MOVL C01429 V=800.0 PL=0
MOVL C01430 V=800.0 PL=0
MOVL C01431 V=800.0 PL=0
MOVL C01432 V=800.0 PL=0
MOVL C01433 V=800.0 PL=0
MOVL C01434 V=800.0 PL=0
MOVL C01435 V=800.0 PL=0
MOVL C01436 V=800.0 PL=0
MOVL C01437 V=800.0 PL=0
MOVL C01438 V=800.0 PL=0
MOVL C01439 V=800.0 PL=0
MOVL C01440 V=800.0 PL=0
MOVL C01441 V=800.0 PL=0
MOVL C01442 V=800.0 PL=0
MOVL C01443 V=800.0 PL=0
MOVL C01444 V=800.0 PL=0
MOVL C01445 V=800.0 PL=0
MOVL C01446 V=800.0 PL=0
MOVL C01447 V=800.0 PL=0
MOVL C01448 V=800.0 PL=0
MOVL C01449 V=800.0 PL=0
MOVL C01450 V=800.0 PL=0
MOVL C01451 V=800.0 PL=0
MOVL C01452 V=800.0 PL=0
MOVL C01453 V=800.0 PL=0
MOVL C01454 V=800.0 PL=0
MOVL C01455 V=800.0 PL=0
MOVL C01456 V=800.0 PL=0
MOVL C01457 V=800.0 PL=0
MOVL C01458 V=800.0 PL=0
MOVL C01459 V=800.0 PL=0
MOVL C01460 V=800.0 PL=0
MOVL C01461 V=800.0 PL=0
MOVL C01462 V=800.0 PL=0
MOVL C01463 V=800.0 PL=0
MOVL C01464 V=800.0 PL=0
MOVL C01465 V=800.0 PL=0
MOVL C01466 V=800.0 PL=0
MOVL C01467 V=800.0 PL=0
MOVL C01468 V=800.0 PL=0
MOVL C01469 V=800.0 PL=0
MOVL C01470 V=800.0 PL=0
MOVL C01471 V=800.0 PL=0
MOVL C01472 V=800.0 PL=0
MOVL C01473 V=800.0 PL=0
MOVL C01474 V=800.0 PL=0
MOVL C01475 V=800.0 PL=0
MOVL C01476 V=800.0 PL=0
MOVL C01477 V=800.0 PL=0
MOVL C01478 V=800.0 PL=0
MOVL C01479 V=800.0 PL=0
MOVL C01480 V=800.0 PL=0
MOVL C01481 V=800.0 PL=0
MOVL C01482 V=800.0 PL=0
MOVL C01483 V=800.0 PL=0
MOVL C01484 V=800.0 PL=0
MOVL C01485 V=800.0 PL=0
MOVL C01486 V=800.0 PL=0
MOVL C01487 V=800.0 PL=0
MOVL C01488 V=800.0 PL=0
MOVL C01489 V=800.0 PL=0
MOVL C01490 V=800.0 PL=0
MOVL C01491 V=800.0 PL=0
MOVL C01492 V=800.0 PL=0
MOVL C01493 V=800.0 PL=0
MOVL C01494 V=800.0 PL=0
MOVL C01495 V=800.0 PL=0
MOVL C01496 V=800.0 PL=0
MOVL C01497 V=800.0 PL=0
MOVL C01498 V=800.0 PL=0
MOVL C01499 V=800.0 PL=0
MOVL C01500 V=800.0 PL=0
MOVL C01501 V=800.0 PL=0
MOVL C01502 V=800.0 PL=0
MOVL C01503 V=800.0 PL=0
MOVL C01504 V=800.0 PL=0
MOVL C01505 V=800.0 PL=0
MOVL C01506 V=800.0 PL=0
MOVL C01507 V=800.0 PL=0
MOVL C01508 V=800.0 PL=0
MOVL C01509 V=800.0 PL=0
MOVL C01510 V=800.0 PL=0
MOVL C01511 V=800.0 PL=0
MOVL C01512 V=800.0 PL=0
MOVL C01513 V=800.0 PL=0
MOVL C01514 V=800.0 PL=0
MOVL C01515 V=800.0 PL=0
MOVL C01516 V=800.0 PL=0
MOVL C01517 V=800.0 PL=0
MOVL C01518 V=800.0 PL=0
MOVL C01519 V=800.0 PL=0
MOVL C01520 V=800.0 PL=0
MOVL C01521 V=800.0 PL=0
MOVL C01522 V=800.0 PL=0
MOVL C01523 V=800.0 PL=0
MOVL C01524 V=800.0 PL=0
MOVL C01525 V=800.0 PL=0
MOVL C01526 V=800.0 PL=0
MOVL C01527 V=800.0 PL=0
MOVL C01528 V=800.0 PL=0
MOVL C01529 V=800.0 PL=0
MOVL C01530 V=800.0 PL=0
MOVL C01531 V=800.0 PL=0
MOVL C01532 V=800.0 PL=0
MOVL C01533 V=800.0 PL=0
MOVL C01534 V=800.0 PL=0
MOVL C01535 V=800.0 PL=0
MOVL C01536 V=800.0 PL=0
MOVL C01537 V=800.0 PL=0
MOVL C01538 V=800.0 PL=0
MOVL C01539 V=800.0 PL=0
MOVL C01540 V=800.0 PL=0
MOVL C01541 V=800.0 PL=0
MOVL C01542 V=800.0 PL=0
MOVL C01543 V=800.0 PL=0
MOVL C01544 V=800.0 PL=0
MOVL C01545 V=800.0 PL=0
MOVL C01546 V=800.0 PL=0
MOVL C01547 V=800.0 PL=0
MOVL C01548 V=800.0 PL=0
MOVL C01549 V=800.0 PL=0
MOVL C01550 V=800.0 PL=0
MOVL C01551 V=800.0 PL=0
MOVL C01552 V=800.0 PL=0
MOVL C01553 V=800.0 PL=0
MOVL C01554 V=800.0 PL=0
MOVL C01555 V=800.0 PL=0
MOVL C01556 V=800.0 PL=0
MOVL C01557 V=800.0 PL=0
MOVL C01558 V=800.0 PL=0
MOVL C01559 V=800.0 PL=0
MOVL C01560 V=800.0 PL=0
MOVL C01561 V=800.0 PL=0
MOVL C01562 V=800.0 PL=0
MOVL C01563 V=800.0 PL=0
MOVL C01564 V=800.0 PL=0
MOVL C01565 V=800.0 PL=0
MOVL C01566 V=800.0 PL=0
MOVL C01567 V=800.0 PL=0
MOVL C01568 V=800.0 PL=0
MOVL C01569 V=800.0 PL=0
MOVL C01570 V=800.0 PL=0
MOVL C01571 V=800.0 PL=0
MOVL C01572 V=800.0 PL=0
MOVL C01573 V=800.0 PL=0
MOVL C01574 V=800.0 PL=0
MOVL C01575 V=800.0 PL=0
MOVL C01576 V=800.0 PL=0
MOVL C01577 V=800.0 PL=0
MOVL C01578 V=800.0 PL=0
MOVL C01579 V=800.0 PL=0
MOVL C01580 V=800.0 PL=0
MOVL C01581 V=800.0 PL=0
MOVL C01582 V=800.0 PL=0
MOVL C01583 V=800.0 PL=0
MOVL C01584 V=800.0 PL=0
MOVL C01585 V=800.0 PL=0
MOVL C01586 V=800.0 PL=0
MOVL C01587 V=800.0 PL=0
MOVL C01588 V=800.0 PL=0
MOVL C01589 V=800.0 PL=0
MOVL C01590 V=800.0 PL=0
MOVL C01591 V=800.0 PL=0
MOVL C01592 V=800.0 PL=0
MOVL C01593 V=800.0 PL=0
MOVL C01594 V=800.0 PL=0
MOVL C01595 V=800.0 PL=0
MOVL C01596 V=800.0 PL=0
MOVL C01597 V=800.0 PL=0
MOVL C01598 V=800.0 PL=0
MOVL C01599 V=800.0 PL=0
MOVL C01600 V=800.0 PL=0
MOVL C01601 V=800.0 PL=0
MOVL C01602 V=800.0 PL=0
MOVL C01603 V=800.0 PL=0
MOVL C01604 V=800.0 PL=0
MOVL C01605 V=800.0 PL=0
MOVL C01606 V=800.0 PL=0
MOVL C01607 V=800.0 PL=0
MOVL C01608 V=800.0 PL=0
MOVL C01609 V=800.0 PL=0
MOVL C01610 V=800.0 PL=0
MOVL C01611 V=800.0 PL=0
MOVL C01612 V=800.0 PL=0
MOVL C01613 V=800.0 PL=0
MOVL C01614 V=800.0 PL=0
MOVL C01615 V=800.0 PL=0
MOVL C01616 V=800.0 PL=0
MOVL C01617 V=800.0 PL=0
MOVL C01618 V=800.0 PL=0
MOVL C01619 V=800.0 PL=0
MOVL C01620 V=800.0 PL=0
MOVL C01621 V=800.0 PL=0
MOVL C01622 V=800.0 PL=0
MOVL C01623 V=800.0 PL=0
MOVL C01624 V=800.0 PL=0
MOVL C01625 V=800.0 PL=0
MOVL C01626 V=800.0 PL=0
MOVL C01627 V=800.0 PL=0
MOVL C01628 V=800.0 PL=0
MOVL C01629 V=800.0 PL=0
MOVL C01630 V=800.0 PL=0
MOVL C01631 V=800.0 PL=0
MOVL C01632 V=800.0 PL=0
MOVL C01633 V=800.0 PL=0
MOVL C01634 V=800.0 PL=0
MOVL C01635 V=800.0 PL=0
MOVL C01636 V=800.0 PL=0
MOVL C01637 V=800.0 PL=0
MOVL C01638 V=800.0 PL=0
MOVL C01639 V=800.0 PL=0
MOVL C01640 V=800.0 PL=0
MOVL C01641 V=800.0 PL=0
MOVL C01642 V=800.0 PL=0
MOVL C01643 V=800.0 PL=0
MOVL C01644 V=800.0 PL=0
MOVL C01645 V=800.0 PL=0
MOVL C01646 V=800.0 PL=0
MOVL C01647 V=800.0 PL=0
MOVL C01648 V=800.0 PL=0
MOVL C01649 V=800.0 PL=0
MOVL C01650 V=800.0 PL=0
MOVL C01651 V=800.0 PL=0
MOVL C01652 V=800.0 PL=0
MOVL C01653 V=800.0 PL=0
MOVL C01654 V=800.0 PL=0
MOVL C01655 V=800.0 PL=0
MOVL C01656 V=800.0 PL=0
MOVL C01657 V=800.0 PL=0
MOVL C01658 V=800.0 PL=0
MOVL C01659 V=800.0 PL=0
MOVL C01660 V=800.0 PL=0
MOVL C01661 V=800.0 PL=0
MOVL C01662 V=800.0 PL=0
MOVL C01663 V=800.0 PL=0
MOVL C01664 V=800.0 PL=0
MOVL C01665 V=800.0 PL=0
MOVL C01666 V=800.0 PL=0
MOVL C01667 V=800.0 PL=0
MOVL C01668 V=800.0 PL=0
MOVL C01669 V=800.0 PL=0
MOVL C01670 V=800.0 PL=0
MOVL C01671 V=800.0 PL=0
MOVL C01672 V=800.0 PL=0
MOVL C01673 V=800.0 PL=0
MOVL C01674 V=800.0 PL=0
MOVL C01675 V=800.0 PL=0
MOVL C01676 V=800.0 PL=0
MOVL C01677 V=800.0 PL=0
MOVL C01678 V=800.0 PL=0
MOVL C01679 V=800.0 PL=0
MOVL C01680 V=800.0 PL=0
MOVL C01681 V=800.0 PL=0
MOVL C01682 V=800.0 PL=0
MOVL C01683 V=800.0 PL=0
MOVL C01684 V=800.0 PL=0
MOVL C01685 V=800.0 PL=0
MOVL C01686 V=800.0 PL=0
MOVL C01687 V=800.0 PL=0
MOVL C01688 V=800.0 PL=0
MOVL C01689 V=800.0 PL=0
MOVL C01690 V=800.0 PL=0
MOVL C01691 V=800.0 PL=0
MOVL C01692 V=800.0 PL=0
MOVL C01693 V=800.0 PL=0
MOVL C01694 V=800.0 PL=0
MOVL C01695 V=800.0 PL=0
MOVL C01696 V=800.0 PL=0
MOVL C01697 V=800.0 PL=0
MOVL C01698 V=800.0 PL=0
MOVL C01699 V=800.0 PL=0
MOVL C01700 V=800.0 PL=0
MOVL C01701 V=800.0 PL=0
MOVL C01702 V=800.0 PL=0
MOVL C01703 V=800.0 PL=0
MOVL C01704 V=800.0 PL=0
MOVL C01705 V=800.0 PL=0
MOVL C01706 V=800.0 PL=0
MOVL C01707 V=800.0 PL=0
MOVL C01708 V=800.0 PL=0
MOVL C01709 V=800.0 PL=0
MOVL C01710 V=800.0 PL=0
MOVL C01711 V=800.0 PL=0
MOVL C01712 V=800.0 PL=0
MOVL C01713 V=800.0 PL=0
MOVL C01714 V=800.0 PL=0
MOVL C01715 V=800.0 PL=0
MOVL C01716 V=800.0 PL=0
MOVL C01717 V=800.0 PL=0
MOVL C01718 V=800.0 PL=0
MOVL C01719 V=800.0 PL=0
MOVL C01720 V=800.0 PL=0
MOVL C01721 V=800.0 PL=0
MOVL C01722 V=800.0 PL=0
MOVL C01723 V=800.0 PL=0
MOVL C01724 V=800.0 PL=0
MOVL C01725 V=800.0 PL=0
MOVL C01726 V=800.0 PL=0
MOVL C01727 V=800.0 PL=0
MOVL C01728 V=800.0 PL=0
MOVL C01729 V=800.0 PL=0
MOVL C01730 V=800.0 PL=0
MOVL C01731 V=800.0 PL=0
MOVL C01732 V=800.0 PL=0
MOVL C01733 V=800.0 PL=0
MOVL C01734 V=800.0 PL=0
MOVL C01735 V=800.0 PL=0
MOVL C01736 V=800.0 PL=0
MOVL C01737 V=800.0 PL=0
MOVL C01738 V=800.0 PL=0
MOVL C01739 V=800.0 PL=0
MOVL C01740 V=800.0 PL=0
MOVL C01741 V=800.0 PL=0
MOVL C01742 V=800.0 PL=0
MOVL C01743 V=800.0 PL=0
MOVL C01744 V=800.0 PL=0
MOVL C01745 V=800.0 PL=0
MOVL C01746 V=800.0 PL=0
MOVL C01747 V=800.0 PL=0
MOVL C01748 V=800.0 PL=0
MOVL C01749 V=800.0 PL=0
MOVL C01750 V=800.0 PL=0
MOVL C01751 V=800.0 PL=0
MOVL C01752 V=800.0 PL=0
MOVL C01753 V=800.0 PL=0
MOVL C01754 V=800.0 PL=0
MOVL C01755 V=800.0 PL=0
MOVL C01756 V=800.0 PL=0
MOVL C01757 V=800.0 PL=0
MOVL C01758 V=800.0 PL=0
MOVL C01759 V=800.0 PL=0
MOVL C01760 V=800.0 PL=0
MOVL C01761 V=800.0 PL=0
MOVL C01762 V=800.0 PL=0
MOVL C01763 V=800.0 PL=0
MOVL C01764 V=800.0 PL=0
MOVL C01765 V=800.0 PL=0
MOVL C01766 V=800.0 PL=0
MOVL C01767 V=800.0 PL=0
MOVL C01768 V=800.0 PL=0
MOVL C01769 V=800.0 PL=0
MOVL C01770 V=800.0 PL=0
MOVL C01771 V=800.0 PL=0
MOVL C01772 V=800.0 PL=0
MOVL C01773 V=800.0 PL=0
MOVL C01774 V=800.0 PL=0
MOVL C01775 V=800.0 PL=0
MOVL C01776 V=800.0 PL=0
MOVL C01777 V=800.0 PL=0
MOVL C01778 V=800.0 PL=0
MOVL C01779 V=800.0 PL=0
MOVL C01780 V=800.0 PL=0
MOVL C01781 V=800.0 PL=0
MOVL C01782 V=800.0 PL=0
MOVL C01783 V=800.0 PL=0
MOVL C01784 V=800.0 PL=0
MOVL C01785 V=800.0 PL=0
MOVL C01786 V=800.0 PL=0
MOVL C01787 V=800.0 PL=0
MOVL C01788 V=800.0 PL=0
MOVL C01789 V=800.0 PL=0
MOVL C01790 V=800.0 PL=0
MOVL C01791 V=800.0 PL=0
MOVL C01792 V=800.0 PL=0
MOVL C01793 V=800.0 PL=0
MOVL C01794 V=800.0 PL=0
MOVL C01795 V=800.0 PL=0
MOVL C01796 V=800.0 PL=0
MOVL C01797 V=800.0 PL=0
MOVL C01798 V=800.0 PL=0
MOVL C01799 V=800.0 PL=0
MOVL C01800 V=800.0 PL=0
MOVL C01801 V=800.0 PL=0
MOVL C01802 V=800.0 PL=0
MOVL C01803 V=800.0 PL=0
MOVL C01804 V=800.0 PL=0
MOVL C01805 V=800.0 PL=0
MOVL C01806 V=800.0 PL=0
MOVL C01807 V=800.0 PL=0
MOVL C01808 V=800.0 PL=0
MOVL C01809 V=800.0 PL=0
MOVL C01810 V=800.0 PL=0
MOVL C01811 V=800.0 PL=0
MOVL C01812 V=800.0 PL=0
MOVL C01813 V=800.0 PL=0
MOVL C01814 V=800.0 PL=0
MOVL C01815 V=800.0 PL=0
MOVL C01816 V=800.0 PL=0
MOVL C01817 V=800.0 PL=0
MOVL C01818 V=800.0 PL=0
MOVL C01819 V=800.0 PL=0
MOVL C01820 V=800.0 PL=0
MOVL C01821 V=800.0 PL=0
MOVL C01822 V=800.0 PL=0
MOVL C01823 V=800.0 PL=0
MOVL C01824 V=800.0 PL=0
MOVL C01825 V=800.0 PL=0
MOVL C01826 V=800.0 PL=0
MOVL C01827 V=800.0 PL=0
MOVL C01828 V=800.0 PL=0
MOVL C01829 V=800.0 PL=0
MOVL C01830 V=800.0 PL=0
MOVL C01831 V=800.0 PL=0
MOVL C01832 V=800.0 PL=0
MOVL C01833 V=800.0 PL=0
MOVL C01834 V=800.0 PL=0
MOVL C01835 V=800.0 PL=0
MOVL C01836 V=800.0 PL=0
MOVL C01837 V=800.0 PL=0
MOVL C01838 V=800.0 PL=0
MOVL C01839 V=800.0 PL=0
MOVL C01840 V=800.0 PL=0
MOVL C01841 V=800.0 PL=0
MOVL C01842 V=800.0 PL=0
MOVL C01843 V=800.0 PL=0
MOVL C01844 V=800.0 PL=0
MOVL C01845 V=800.0 PL=0
MOVL C01846 V=800.0 PL=0
MOVL C01847 V=800.0 PL=0
MOVL C01848 V=800.0 PL=0
MOVL C01849 V=800.0 PL=0
MOVL C01850 V=800.0 PL=0
MOVL C01851 V=800.0 PL=0
MOVL C01852 V=800.0 PL=0
MOVL C01853 V=800.0 PL=0
MOVL C01854 V=800.0 PL=0
MOVL C01855 V=800.0 PL=0
MOVL C01856 V=800.0 PL=0
MOVL C01857 V=800.0 PL=0
MOVL C01858 V=800.0 PL=0
MOVL C01859 V=800.0 PL=0
MOVL C01860 V=800.0 PL=0
MOVL C01861 V=800.0 PL=0
MOVL C01862 V=800.0 PL=0
MOVL C01863 V=800.0 PL=0
MOVL C01864 V=800.0 PL=0
MOVL C01865 V=800.0 PL=0
MOVL C01866 V=800.0 PL=0
MOVL C01867 V=800.0 PL=0
MOVL C01868 V=800.0 PL=0
MOVL C01869 V=800.0 PL=0
MOVL C01870 V=800.0 PL=0
MOVL C01871 V=800.0 PL=0
MOVL C01872 V=800.0 PL=0
MOVL C01873 V=800.0 PL=0
MOVL C01874 V=800.0 PL=0
MOVL C01875 V=800.0 PL=0
MOVL C01876 V=800.0 PL=0
MOVL C01877 V=800.0 PL=0
MOVL C01878 V=800.0 PL=0
MOVL C01879 V=800.0 PL=0
MOVL C01880 V=800.0 PL=0
MOVL C01881 V=800.0 PL=0
MOVL C01882 V=800.0 PL=0
MOVL C01883 V=800.0 PL=0
MOVL C01884 V=800.0 PL=0
MOVL C01885 V=800.0 PL=0
MOVL C01886 V=800.0 PL=0
MOVL C01887 V=800.0 PL=0
MOVL C01888 V=800.0 PL=0
MOVL C01889 V=800.0 PL=0
MOVL C01890 V=800.0 PL=0
MOVL C01891 V=800.0 PL=0
MOVL C01892 V=800.0 PL=0
MOVL C01893 V=800.0 PL=0
MOVL C01894 V=800.0 PL=0
MOVL C01895 V=800.0 PL=0
MOVL C01896 V=800.0 PL=0
MOVL C01897 V=800.0 PL=0
MOVL C01898 V=800.0 PL=0
MOVL C01899 V=800.0 PL=0
MOVL C01900 V=800.0 PL=0
MOVL C01901 V=800.0 PL=0
MOVL C01902 V=800.0 PL=0
MOVL C01903 V=800.0 PL=0
MOVL C01904 V=800.0 PL=0
MOVL C01905 V=800.0 PL=0
MOVL C01906 V=800.0 PL=0
MOVL C01907 V=800.0 PL=0
MOVL C01908 V=800.0 PL=0
MOVL C01909 V=800.0 PL=0
MOVL C01910 V=800.0 PL=0
MOVL C01911 V=800.0 PL=0
MOVL C01912 V=800.0 PL=0
MOVL C01913 V=800.0 PL=0
MOVL C01914 V=800.0 PL=0
MOVL C01915 V=800.0 PL=0
MOVL C01916 V=800.0 PL=0
MOVL C01917 V=800.0 PL=0
MOVL C01918 V=800.0 PL=0
MOVL C01919 V=800.0 PL=0
MOVL C01920 V=800.0 PL=0
MOVL C01921 V=800.0 PL=0
MOVL C01922 V=800.0 PL=0
MOVL C01923 V=800.0 PL=0
MOVL C01924 V=800.0 PL=0
MOVL C01925 V=800.0 PL=0
MOVL C01926 V=800.0 PL=0
MOVL C01927 V=800.0 PL=0
MOVL C01928 V=800.0 PL=0
MOVL C01929 V=800.0 PL=0
MOVL C01930 V=800.0 PL=0
MOVL C01931 V=800.0 PL=0
MOVL C01932 V=800.0 PL=0
MOVL C01933 V=800.0 PL=0
MOVL C01934 V=800.0 PL=0
MOVL C01935 V=800.0 PL=0
MOVL C01936 V=800.0 PL=0
MOVL C01937 V=800.0 PL=0
MOVL C01938 V=800.0 PL=0
MOVL C01939 V=800.0 PL=0
MOVL C01940 V=800.0 PL=0
MOVL C01941 V=800.0 PL=0
MOVL C01942 V=800.0 PL=0
MOVL C01943 V=800.0 PL=0
MOVL C01944 V=800.0 PL=0
MOVL C01945 V=800.0 PL=0
MOVL C01946 V=800.0 PL=0
MOVL C01947 V=800.0 PL=0
MOVL C01948 V=800.0 PL=0
MOVL C01949 V=800.0 PL=0
MOVL C01950 V=800.0 PL=0
MOVL C01951 V=800.0 PL=0
MOVL C01952 V=800.0 PL=0
MOVL C01953 V=800.0 PL=0
MOVL C01954 V=800.0 PL=0
MOVL C01955 V=800.0 PL=0
MOVL C01956 V=800.0 PL=0
MOVL C01957 V=800.0 PL=0
MOVL C01958 V=800.0 PL=0
MOVL C01959 V=800.0 PL=0
MOVL C01960 V=800.0 PL=0
MOVL C01961 V=800.0 PL=0
MOVL C01962 V=800.0 PL=0
MOVL C01963 V=800.0 PL=0
MOVL C01964 V=800.0 PL=0
MOVL C01965 V=800.0 PL=0
MOVL C01966 V=800.0 PL=0
MOVL C01967 V=800.0 PL=0
MOVL C01968 V=800.0 PL=0
MOVL C01969 V=800.0 PL=0
MOVL C01970 V=800.0 PL=0
MOVL C01971 V=800.0 PL=0
MOVL C01972 V=800.0 PL=0
MOVL C01973 V=800.0 PL=0
MOVL C01974 V=800.0 PL=0
MOVL C01975 V=800.0 PL=0
MOVL C01976 V=800.0 PL=0
MOVL C01977 V=800.0 PL=0
MOVL C01978 V=800.0 PL=0
MOVL C01979 V=800.0 PL=0
MOVL C01980 V=800.0 PL=0
MOVL C01981 V=800.0 PL=0
MOVL C01982 V=800.0 PL=0
MOVL C01983 V=800.0 PL=0
MOVL C01984 V=800.0 PL=0
MOVL C01985 V=800.0 PL=0
MOVL C01986 V=800.0 PL=0
MOVL C01987 V=800.0 PL=0
MOVL C01988 V=800.0 PL=0
MOVL C01989 V=800.0 PL=0
MOVL C01990 V=800.0 PL=0
MOVL C01991 V=800.0 PL=0
MOVL C01992 V=800.0 PL=0
MOVL C01993 V=800.0 PL=0
MOVL C01994 V=800.0 PL=0
MOVL C01995 V=800.0 PL=0
MOVL C01996 V=800.0 PL=0
MOVL C01997 V=800.0 PL=0
MOVL C01998 V=800.0 PL=0
MOVL C01999 V=800.0 PL=0
MOVL C02000 V=800.0 PL=0
MOVL C02001 V=800.0 PL=0
MOVL C02002 V=800.0 PL=0
MOVL C02003 V=800.0 PL=0
MOVL C02004 V=800.0 PL=0
MOVL C02005 V=800.0 PL=0
MOVL C02006 V=800.0 PL=0
MOVL C02007 V=800.0 PL=0
MOVL C02008 V=800.0 PL=0
MOVL C02009 V=800.0 PL=0
MOVL C02010 V=800.0 PL=0
MOVL C02011 V=800.0 PL=0
MOVL C02012 V=800.0 PL=0
MOVL C02013 V=800.0 PL=0
MOVL C02014 V=800.0 PL=0
MOVL C02015 V=800.0 PL=0
MOVL C02016 V=800.0 PL=0
MOVL C02017 V=800.0 PL=0
MOVL C02018 V=800.0 PL=0
MOVL C02019 V=800.0 PL=0
MOVL C02020 V=800.0 PL=0
MOVL C02021 V=800.0 PL=0
MOVL C02022 V=800.0 PL=0
MOVL C02023 V=800.0 PL=0
MOVL C02024 V=800.0 PL=0
MOVL C02025 V=800.0 PL=0
MOVL C02026 V=800.0 PL=0
MOVL C02027 V=800.0 PL=0
MOVL C02028 V=800.0 PL=0
MOVL C02029 V=800.0 PL=0
MOVL C02030 V=800.0 PL=0
MOVL C02031 V=800.0 PL=0
MOVL C02032 V=800.0 PL=0
MOVL C02033 V=800.0 PL=0
MOVL C02034 V=800.0 PL=0
MOVL C02035 V=800.0 PL=0
MOVL C02036 V=800.0 PL=0
MOVL C02037 V=800.0 PL=0
MOVL C02038 V=800.0 PL=0
MOVL C02039 V=800.0 PL=0
MOVL C02040 V=800.0 PL=0
MOVL C02041 V=800.0 PL=0
MOVL C02042 V=800.0 PL=0
MOVL C02043 V=800.0 PL=0
MOVL C02044 V=800.0 PL=0
MOVL C02045 V=800.0 PL=0
MOVL C02046 V=800.0 PL=0
MOVL C02047 V=800.0 PL=0
MOVL C02048 V=800.0 PL=0
MOVL C02049 V=800.0 PL=0
MOVL C02050 V=800.0 PL=0
MOVL C02051 V=800.0 PL=0
MOVL C02052 V=800.0 PL=0
MOVL C02053 V=800.0 PL=0
MOVL C02054 V=800.0 PL=0
MOVL C02055 V=800.0 PL=0
MOVL C02056 V=800.0 PL=0
MOVL C02057 V=800.0 PL=0
MOVL C02058 V=800.0 PL=0
MOVL C02059 V=800.0 PL=0
MOVL C02060 V=800.0 PL=0
MOVL C02061 V=800.0 PL=0
MOVL C02062 V=800.0 PL=0
MOVL C02063 V=800.0 PL=0
MOVL C02064 V=800.0 PL=0
MOVL C02065 V=800.0 PL=0
MOVL C02066 V=800.0 PL=0
MOVL C02067 V=800.0 PL=0
MOVL C02068 V=800.0 PL=0
MOVL C02069 V=800.0 PL=0
MOVL C02070 V=800.0 PL=0
MOVL C02071 V=800.0 PL=0
MOVL C02072 V=800.0 PL=0
MOVL C02073 V=800.0 PL=0
MOVL C02074 V=800.0 PL=0
MOVL C02075 V=800.0 PL=0
MOVL C02076 V=800.0 PL=0
MOVL C02077 V=800.0 PL=0
MOVL C02078 V=800.0 PL=0
